C01833=1202.027,168.562,-55.131,-177.976,6.217,148.523
C01834=1202.022,168.811,-55.153,-177.973,6.219,148.522
C01835=1202.018,169.060,-55.175,-177.970,6.220,148.522
C01836=1202.013,169.309,-55.197,-177.968,6.222,148.522
C01837=1202.008,169.559,-55.219,-177.965,6.224,148.521
C01838=1202.003,169.807,-55.241,-177.963,6.225,148.521
C01839=1201.999,170.056,-55.263,-177.960,6.227,148.521
C01840=1201.994,170.305,-55.286,-177.957,6.228,148.520
C01841=1201.990,170.554,-55.308,-177.954,6.230,148.520
C01842=1201.985,170.803,-55.329,-177.952,6.232,148.519
C01843=1201.980,171.052,-55.351,-177.950,6.233,148.519
C01844=1201.975,171.301,-55.374,-177.947,6.235,148.518
C01845=1201.971,171.550,-55.396,-177.944,6.236,148.518
C01846=1201.967,171.799,-55.419,-177.942,6.238,148.518
C01847=1201.962,172.048,-55.440,-177.939,6.240,148.517
C01848=1201.957,172.297,-55.464,-177.936,6.242,148.517
C01849=1201.952,172.546,-55.485,-177.934,6.242,148.516
C01850=1201.948,172.795,-55.507,-177.931,6.244,148.516
C01851=1201.942,173.044,-55.530,-177.928,6.246,148.516
C01852=1201.938,173.293,-55.552,-177.926,6.248,148.515
C01853=1201.934,173.542,-55.574,-177.923,6.250,148.515
C01854=1201.928,173.791,-55.597,-177.920,6.251,148.515
C01855=1201.924,174.040,-55.619,-177.918,6.252,148.514
C01856=1201.920,174.288,-55.641,-177.916,6.254,148.514
C01857=1201.915,174.538,-55.664,-177.913,6.256,148.513
C01858=1201.911,174.787,-55.687,-177.910,6.258,148.513
C01859=1201.906,175.035,-55.708,-177.907,6.259,148.513
C01860=1201.901,175.284,-55.732,-177.904,6.261,148.512
C01861=1201.897,175.534,-55.754,-177.902,6.262,148.512
C01862=1201.891,175.783,-55.776,-177.900,6.264,148.511
C01863=1201.887,176.031,-55.799,-177.897,6.266,148.511
C01864=1201.882,176.280,-55.820,-177.894,6.268,148.511
C01865=1201.878,176.529,-55.844,-177.892,6.269,148.510
C01866=1201.873,176.778,-55.866,-177.889,6.271,148.510
C01867=1201.868,177.027,-55.889,-177.886,6.273,148.510
C01868=1201.864,177.276,-55.911,-177.884,6.274,148.509
C01869=1201.860,177.525,-55.934,-177.882,6.276,148.509
C01870=1201.854,177.774,-55.956,-177.879,6.278,148.509
C01871=1201.850,178.022,-55.979,-177.876,6.279,148.508
C01872=1201.845,178.272,-56.001,-177.873,6.281,148.508
C01873=1201.841,178.520,-56.024,-177.870,6.283,148.507
C01874=1201.836,178.770,-56.046,-177.868,6.284,148.507
C01875=1201.832,179.018,-56.069,-177.866,6.285,148.506
C01876=1201.827,179.268,-56.092,-177.863,6.287,148.506
C01877=1201.822,179.516,-56.114,-177.860,6.289,148.506
C01878=1201.818,179.765,-56.137,-177.858,6.291,148.505
C01879=1201.813,180.014,-56.159,-177.855,6.293,148.505
C01880=1201.808,180.263,-56.182,-177.852,6.294,148.505
C01881=1201.804,180.512,-56.205,-177.850,6.296,148.504
C01882=1201.799,180.761,-56.228,-177.847,6.298,148.504
C01883=1201.795,181.010,-56.251,-177.844,6.300,148.504
C01884=1201.789,181.259,-56.273,-177.842,6.301,148.503
C01885=1201.785,181.508,-56.296,-177.840,6.303,148.503
C01886=1201.781,181.757,-56.319,-177.837,6.304,148.503
C01887=1201.776,182.006,-56.342,-177.834,6.306,148.502
C01888=1201.771,182.254,-56.364,-177.832,6.308,148.502
C01889=1201.766,182.503,-56.387,-177.829,6.310,148.501
C01890=1201.763,182.752,-56.410,-177.826,6.312,148.501
C01891=1201.758,183.002,-56.433,-177.824,6.313,148.501
C01892=1201.752,183.250,-56.456,-177.821,6.315,148.500
C01893=1201.748,183.499,-56.479,-177.818,6.316,148.500
C01894=1201.743,183.748,-56.501,-177.816,6.318,148.499
C01895=1201.739,183.997,-56.524,-177.813,6.320,148.499
C01896=1201.735,184.246,-56.547,-177.810,6.321,148.499
C01897=1201.729,184.494,-56.570,-177.808,6.323,148.498
C01898=1201.725,184.764,-56.595,-177.805,6.325,148.498
C01899=1201.719,185.034,-56.620,-177.802,6.327,148.498
C01900=1201.715,185.303,-56.644,-177.799,6.329,148.497
C01901=1201.709,185.573,-56.669,-177.797,6.331,148.497
C01902=1201.705,185.822,-56.693,-177.794,6.333,148.497
C01903=1201.701,186.071,-56.715,-177.791,6.335,148.496
C01904=1201.696,186.320,-56.739,-177.789,6.336,148.496
C01905=1201.691,186.569,-56.762,-177.787,6.338,148.496
C01906=1201.686,186.817,-56.785,-177.784,6.339,148.495
C01907=1201.682,187.066,-56.807,-177.781,6.341,148.495
C01908=1201.677,187.315,-56.831,-177.778,6.343,148.494
C01909=1201.672,187.564,-56.854,-177.775,6.345,148.494
C01910=1201.668,187.813,-56.877,-177.773,6.346,148.494
C01911=1201.664,188.062,-56.900,-177.770,6.348,148.493
C01912=1201.659,188.311,-56.923,-177.767,6.350,148.493
C01913=1201.654,188.560,-56.946,-177.765,6.352,148.493
C01914=1201.649,188.809,-56.970,-177.762,6.354,148.492
C01915=1201.645,189.057,-56.993,-177.760,6.356,148.492
C01916=1201.640,189.306,-57.016,-177.757,6.358,148.492
C01917=1201.636,189.555,-57.039,-177.755,6.359,148.491
C01918=1201.631,189.804,-57.063,-177.752,6.361,148.491
C01919=1201.626,190.053,-57.086,-177.750,6.362,148.491
C01920=1201.622,190.302,-57.109,-177.747,6.364,148.490
C01921=1201.618,190.551,-57.132,-177.745,6.366,148.490
C01922=1201.612,190.800,-57.155,-177.742,6.368,148.490
C01923=1201.608,191.049,-57.178,-177.739,6.369,148.489
C01924=1201.603,191.298,-57.202,-177.737,6.371,148.489
C01925=1201.599,191.546,-57.226,-177.734,6.373,148.488
C01926=1201.595,191.795,-57.249,-177.731,6.375,148.488
C01927=1201.590,192.044,-57.272,-177.729,6.377,148.488
C01928=1201.585,192.293,-57.295,-177.726,6.378,148.487
C01929=1201.581,192.542,-57.319,-177.723,6.380,148.487
C01930=1201.576,192.791,-57.342,-177.721,6.382,148.487
C01931=1201.571,193.040,-57.365,-177.718,6.384,148.486
C01932=1201.567,193.288,-57.389,-177.715,6.386,148.486
C01933=1201.562,193.537,-57.413,-177.713,6.388,148.486
C01934=1201.557,193.786,-57.436,-177.710,6.389,148.485
C01935=1201.553,194.035,-57.459,-177.707,6.391,148.485
C01936=1201.549,194.284,-57.482,-177.705,6.393,148.485
C01937=1201.544,194.533,-57.506,-177.702,6.395,148.484
C01938=1201.540,194.782,-57.530,-177.699,6.397,148.484
C01939=1201.535,195.031,-57.553,-177.697,6.398,148.484
C01940=1201.530,195.280,-57.576,-177.694,6.400,148.483
C01941=1201.526,195.528,-57.601,-177.691,6.402,148.483
C01942=1201.521,195.777,-57.624,-177.689,6.404,148.483
C01943=1201.516,196.026,-57.647,-177.686,6.406,148.482
C01944=1201.512,196.275,-57.671,-177.683,6.408,148.482
C01945=1201.507,196.524,-57.695,-177.681,6.409,148.482
C01946=1201.503,196.773,-57.718,-177.679,6.411,148.481
C01947=1201.498,197.021,-57.742,-177.676,6.413,148.481
C01948=1201.493,197.270,-57.765,-177.673,6.415,148.481
C01949=1201.489,197.519,-57.789,-177.671,6.417,148.480
C01950=1201.484,197.768,-57.813,-177.668,6.419,148.480
C01951=1201.480,198.017,-57.836,-177.665,6.421,148.480
C01952=1201.475,198.266,-57.860,-177.663,6.422,148.479
C01953=1201.471,198.514,-57.884,-177.660,6.424,148.479
C01954=1201.466,198.763,-57.907,-177.657,6.426,148.479
C01955=1201.461,199.011,-57.931,-177.655,6.428,148.478
C01956=1201.456,199.261,-57.955,-177.652,6.430,148.478
C01957=1201.452,199.509,-57.979,-177.649,6.431,148.478
C01958=1201.447,199.758,-58.003,-177.647,6.433,148.477
C01959=1201.443,200.007,-58.027,-177.644,6.435,148.477
C01960=1201.438,200.256,-58.050,-177.641,6.437,148.477
C01961=1201.433,200.505,-58.073,-177.639,6.439,148.476
C01962=1201.429,200.754,-58.098,-177.637,6.441,148.476
C01963=1201.425,201.002,-58.122,-177.634,6.443,148.476
C01964=1201.420,201.251,-58.145,-177.631,6.445,148.475
C01965=1201.415,201.500,-58.170,-177.629,6.446,148.475
C01966=1201.410,201.749,-58.193,-177.626,6.448,148.475
C01967=1201.406,201.997,-58.217,-177.623,6.450,148.474
C01968=1201.401,202.246,-58.241,-177.621,6.452,148.474
C01969=1201.397,202.495,-58.265,-177.618,6.454,148.474
C01970=1201.392,202.744,-58.288,-177.615,6.455,148.473
C01971=1201.388,202.993,-58.313,-177.613,6.458,148.473
C01972=1201.383,203.242,-58.337,-177.611,6.459,148.473
C01973=1201.379,203.491,-58.361,-177.608,6.461,148.473
C01974=1201.374,203.739,-58.385,-177.605,6.463,148.472
C01975=1201.370,203.988,-58.409,-177.603,6.465,148.472
C01976=1201.364,204.237,-58.433,-177.600,6.467,148.472
C01977=1201.360,204.485,-58.457,-177.597,6.469,148.471
C01978=1201.356,204.734,-58.481,-177.595,6.470,148.471
C01979=1201.352,204.983,-58.505,-177.592,6.472,148.471
C01980=1201.346,205.232,-58.529,-177.589,6.474,148.470
C01981=1201.342,205.481,-58.553,-177.587,6.476,148.470
C01982=1201.338,205.729,-58.577,-177.585,6.478,148.470
C01983=1201.334,205.979,-58.601,-177.582,6.480,148.469
C01984=1201.328,206.228,-58.626,-177.579,6.482,148.469
C01985=1201.324,206.476,-58.650,-177.576,6.484,148.469
C01986=1201.320,206.724,-58.674,-177.573,6.486,148.468
C01987=1201.314,206.974,-58.698,-177.571,6.488,148.468
C01988=1201.310,207.223,-58.722,-177.568,6.490,148.468
C01989=1201.306,207.471,-58.746,-177.566,6.492,148.468
C01990=1201.301,207.720,-58.771,-177.563,6.494,148.467
C01991=1201.296,207.968,-58.795,-177.561,6.496,148.467
C01992=1201.292,208.217,-58.818,-177.558,6.497,148.467
C01993=1201.287,208.467,-58.844,-177.555,6.499,148.466
C01994=1201.283,208.715,-58.868,-177.553,6.501,148.466
C01995=1201.278,208.964,-58.892,-177.550,6.503,148.466
C01996=1201.273,209.212,-58.916,-177.548,6.505,148.465
C01997=1201.269,209.461,-58.941,-177.545,6.507,148.465
C01998=1201.264,209.710,-58.965,-177.543,6.509,148.465
C01999=1201.260,209.959,-58.990,-177.539,6.511,148.464
C02000=1201.256,210.207,-59.014,-177.537,6.513,148.464
C02001=1201.251,210.456,-59.039,-177.534,6.515,148.464
C02002=1201.246,210.727,-59.065,-177.531,6.517,148.463
C02003=1201.241,210.997,-59.091,-177.529,6.519,148.463
C02004=1201.236,211.267,-59.117,-177.526,6.521,148.463
C02005=1201.231,211.538,-59.145,-177.523,6.523,148.462
C02006=1201.226,211.787,-59.169,-177.520,6.525,148.462
C02007=1201.222,212.035,-59.193,-177.518,6.527,148.462
C02008=1201.218,212.284,-59.218,-177.516,6.529,148.462
C02009=1201.213,212.533,-59.242,-177.512,6.532,148.461
C02010=1201.209,212.781,-59.266,-177.510,6.533,148.461
C02011=1201.204,213.031,-59.291,-177.507,6.535,148.461
C02012=1201.200,213.279,-59.316,-177.504,6.537,148.460
C02013=1201.195,213.528,-59.340,-177.502,6.539,148.460
C02014=1201.190,213.776,-59.364,-177.500,6.541,148.460
C02015=1201.186,214.026,-59.389,-177.497,6.543,148.460
C02016=1201.181,214.275,-59.414,-177.494,6.545,148.459
C02017=1201.177,214.524,-59.438,-177.492,6.546,148.459
C02018=1201.172,214.772,-59.464,-177.489,6.549,148.459
C02019=1201.167,215.020,-59.488,-177.486,6.551,148.459
C02020=1201.163,215.270,-59.513,-177.484,6.553,148.458
C02021=1201.159,215.518,-59.537,-177.481,6.555,148.458
C02022=1201.153,215.767,-59.562,-177.478,6.557,148.457
C02023=1201.150,216.016,-59.586,-177.476,6.559,148.457
C02024=1201.145,216.264,-59.612,-177.473,6.561,148.457
C02025=1201.140,216.513,-59.637,-177.471,6.563,148.457
C02026=1201.136,216.762,-59.661,-177.468,6.564,148.456
C02027=1201.131,217.011,-59.685,-177.465,6.567,148.456
C02028=1201.127,217.259,-59.710,-177.462,6.569,148.456
C02029=1201.122,217.508,-59.735,-177.460,6.571,148.456
C02030=1201.118,217.757,-59.760,-177.458,6.573,148.455
C02031=1201.113,218.006,-59.784,-177.455,6.575,148.455
C02032=1201.108,218.254,-59.810,-177.452,6.577,148.455
C02033=1201.104,218.503,-59.835,-177.450,6.578,148.454
C02034=1201.099,218.752,-59.859,-177.447,6.581,148.454
C02035=1201.095,219.000,-59.884,-177.444,6.583,148.454
C02036=1201.090,219.249,-59.909,-177.442,6.585,148.454
C02037=1201.086,219.498,-59.934,-177.439,6.587,148.453
C02038=1201.081,219.746,-59.959,-177.437,6.589,148.453
C02039=1201.076,219.995,-59.984,-177.434,6.591,148.453
C02040=1201.073,220.244,-60.009,-177.432,6.593,148.452
C02041=1201.068,220.492,-60.033,-177.429,6.595,148.452
C02042=1201.063,220.742,-60.058,-177.426,6.597,148.452
C02043=1201.058,220.990,-60.084,-177.424,6.599,148.452
C02044=1201.055,221.239,-60.108,-177.421,6.601,148.451
C02045=1201.050,221.487,-60.134,-177.418,6.603,148.451
C02046=1201.045,221.736,-60.159,-177.416,6.605,148.451
C02047=1201.040,221.985,-60.184,-177.413,6.607,148.451
C02048=1201.037,222.234,-60.209,-177.411,6.609,148.450
C02049=1201.032,222.482,-60.234,-177.408,6.611,148.450
C02050=1201.027,222.731,-60.259,-177.405,6.613,148.450
C02051=1201.022,222.979,-60.284,-177.403,6.615,148.450
C02052=1201.019,223.228,-60.309,-177.400,6.617,148.449
C02053=1201.014,223.476,-60.334,-177.397,6.619,148.449
C02054=1201.009,223.726,-60.359,-177.395,6.621,148.449
C02055=1201.004,223.974,-60.385,-177.392,6.624,148.449
C02056=1201.000,224.223,-60.410,-177.389,6.626,148.448
C02057=1200.995,224.472,-60.435,-177.387,6.628,148.448
C02058=1200.992,224.720,-60.460,-177.384,6.629,148.448
C02059=1200.987,224.969,-60.485,-177.382,6.632,148.447
C02060=1200.982,225.218,-60.511,-177.379,6.633,148.447
C02061=1200.978,225.467,-60.536,-177.376,6.636,148.447
C02062=1200.973,225.715,-60.561,-177.374,6.638,148.447
C02063=1200.969,225.964,-60.587,-177.371,6.640,148.446
C02064=1200.964,226.213,-60.611,-177.369,6.642,148.446
C02065=1200.959,226.461,-60.637,-177.366,6.644,148.446
C02066=1200.954,226.710,-60.663,-177.364,6.646,148.446
C02067=1200.951,226.959,-60.687,-177.361,6.649,148.445
C02068=1200.946,227.207,-60.713,-177.358,6.650,148.445
C02069=1200.942,227.456,-60.738,-177.356,6.653,148.445
C02070=1200.937,227.704,-60.764,-177.353,6.654,148.445
C02071=1200.932,227.953,-60.789,-177.351,6.656,148.444
C02072=1200.928,228.202,-60.814,-177.348,6.658,148.444
C02073=1200.924,228.451,-60.840,-177.345,6.661,148.444
C02074=1200.919,228.699,-60.865,-177.343,6.663,148.443
C02075=1200.914,228.948,-60.891,-177.340,6.665,148.443
C02076=1200.910,229.197,-60.916,-177.338,6.667,148.443
C02077=1200.905,229.445,-60.942,-177.335,6.669,148.443
C02078=1200.901,229.694,-60.967,-177.332,6.671,148.442
C02079=1200.896,229.942,-60.993,-177.330,6.674,148.442
C02080=1200.892,230.191,-61.019,-177.327,6.675,148.442
C02081=1200.888,230.440,-61.044,-177.325,6.677,148.442
C02082=1200.883,230.688,-61.069,-177.322,6.679,148.442
C02083=1200.879,230.937,-61.095,-177.319,6.682,148.441
C02084=1200.874,231.186,-61.120,-177.317,6.684,148.441
C02085=1200.870,231.434,-61.146,-177.314,6.686,148.441
C02086=1200.865,231.683,-61.172,-177.312,6.688,148.441
C02087=1200.861,231.932,-61.197,-177.309,6.690,148.440
C02088=1200.856,232.180,-61.223,-177.306,6.693,148.440
C02089=1200.852,232.429,-61.248,-177.304,6.695,148.440
C02090=1200.847,232.678,-61.275,-177.301,6.696,148.440
C02091=1200.842,232.926,-61.300,-177.299,6.699,148.439
C02092=1200.838,233.175,-61.326,-177.296,6.700,148.439
C02093=1200.834,233.423,-61.352,-177.293,6.703,148.439
C02094=1200.830,233.672,-61.377,-177.291,6.705,148.439
C02095=1200.825,233.920,-61.403,-177.288,6.707,148.438
C02096=1200.821,234.169,-61.429,-177.286,6.709,148.438
C02097=1200.816,234.418,-61.454,-177.284,6.711,148.438
C02098=1200.811,234.666,-61.480,-177.280,6.714,148.438
C02099=1200.807,234.915,-61.506,-177.278,6.716,148.437
C02100=1200.802,235.164,-61.532,-177.276,6.718,148.437
C02101=1200.798,235.413,-61.558,-177.273,6.720,148.437
C02102=1200.793,235.661,-61.583,-177.270,6.722,148.437
C02103=1200.789,235.910,-61.609,-177.268,6.724,148.437
C02104=1200.784,236.159,-61.635,-177.265,6.726,148.436
C02105=1200.780,236.408,-61.661,-177.263,6.728,148.436
C02106=1200.775,236.678,-61.689,-177.260,6.731,148.436
C02107=1200.770,236.950,-61.717,-177.257,6.733,148.436
C02108=1200.766,237.221,-61.746,-177.254,6.736,148.435
C02109=1200.760,237.493,-61.774,-177.251,6.738,148.435
C02110=1200.755,237.742,-61.800,-177.248,6.741,148.435
C02111=1200.751,237.990,-61.826,-177.246,6.742,148.435
C02112=1200.747,238.239,-61.852,-177.244,6.745,148.434
C02113=1200.742,238.488,-61.879,-177.241,6.746,148.434
C02114=1200.738,238.736,-61.904,-177.238,6.749,148.434
C02115=1200.733,238.985,-61.930,-177.236,6.751,148.434
C02116=1200.729,239.233,-61.956,-177.233,6.753,148.433
C02117=1200.724,239.482,-61.983,-177.231,6.755,148.433
C02118=1200.720,239.731,-62.008,-177.228,6.758,148.433
C02119=1200.716,239.978,-62.034,-177.225,6.760,148.433
C02120=1200.711,240.227,-62.061,-177.223,6.762,148.433
C02121=1200.707,240.476,-62.086,-177.220,6.764,148.432
C02122=1200.703,240.724,-62.113,-177.218,6.767,148.432
C02123=1200.698,240.974,-62.139,-177.215,6.769,148.432
C02124=1200.693,241.222,-62.165,-177.212,6.770,148.432
C02125=1200.690,241.471,-62.192,-177.210,6.773,148.432
C02126=1200.684,241.719,-62.217,-177.207,6.775,148.431
C02127=1200.680,241.968,-62.243,-177.205,6.777,148.431
C02128=1200.675,242.216,-62.270,-177.202,6.779,148.431
C02129=1200.671,242.465,-62.296,-177.200,6.781,148.431
C02130=1200.667,242.713,-62.323,-177.197,6.784,148.430
C02131=1200.662,242.962,-62.349,-177.194,6.786,148.430
C02132=1200.658,243.211,-62.375,-177.192,6.788,148.430
C02133=1200.653,243.460,-62.402,-177.189,6.791,148.430
C02134=1200.648,243.708,-62.427,-177.187,6.793,148.430
C02135=1200.644,243.956,-62.454,-177.184,6.795,148.429
C02136=1200.639,244.205,-62.480,-177.182,6.797,148.429
C02137=1200.635,244.453,-62.506,-177.179,6.800,148.429
C02138=1200.631,244.702,-62.533,-177.177,6.802,148.429
C02139=1200.627,244.951,-62.559,-177.174,6.804,148.429
C02140=1200.622,245.199,-62.586,-177.171,6.806,148.428
C02141=1200.618,245.448,-62.612,-177.169,6.809,148.428
C02142=1200.613,245.696,-62.639,-177.166,6.810,148.428
C02143=1200.609,245.945,-62.665,-177.164,6.813,148.428
C02144=1200.604,246.194,-62.692,-177.161,6.815,148.427
C02145=1200.600,246.442,-62.718,-177.158,6.817,148.427
C02146=1200.595,246.691,-62.745,-177.156,6.819,148.427
C02147=1200.591,246.939,-62.771,-177.153,6.822,148.427
C02148=1200.586,247.188,-62.797,-177.150,6.824,148.427
C02149=1200.582,247.436,-62.824,-177.148,6.826,148.427
C02150=1200.578,247.685,-62.851,-177.146,6.828,148.426
C02151=1200.573,247.933,-62.876,-177.143,6.831,148.426
C02152=1200.568,248.181,-62.903,-177.140,6.833,148.426
C02153=1200.564,248.430,-62.930,-177.138,6.835,148.426
C02154=1200.559,248.679,-62.956,-177.135,6.838,148.426
C02155=1200.555,248.927,-62.983,-177.132,6.840,148.425
C02156=1200.551,249.175,-63.010,-177.130,6.842,148.425
C02157=1200.546,249.424,-63.037,-177.127,6.844,148.425
C02158=1200.541,249.673,-63.063,-177.125,6.847,148.425
C02159=1200.537,249.921,-63.090,-177.122,6.848,148.424
C02160=1200.533,250.170,-63.117,-177.120,6.851,148.424
C02161=1200.529,250.419,-63.144,-177.117,6.853,148.424
C02162=1200.525,250.667,-63.171,-177.115,6.855,148.424
C02163=1200.520,250.916,-63.197,-177.112,6.858,148.424
C02164=1200.516,251.164,-63.223,-177.109,6.860,148.424
C02165=1200.511,251.413,-63.250,-177.107,6.862,148.423
C02166=1200.506,251.661,-63.278,-177.104,6.865,148.423
C02167=1200.502,251.910,-63.305,-177.101,6.867,148.423
C02168=1200.498,252.158,-63.331,-177.099,6.869,148.423
C02169=1200.493,252.407,-63.358,-177.097,6.872,148.423
C02170=1200.488,252.656,-63.384,-177.094,6.874,148.423
C02171=1200.484,252.904,-63.411,-177.092,6.876,148.422
C02172=1200.480,253.152,-63.438,-177.089,6.879,148.422
C02173=1200.475,253.401,-63.465,-177.086,6.881,148.422
C02174=1200.470,253.649,-63.492,-177.084,6.883,148.422
C02175=1200.466,253.898,-63.519,-177.081,6.886,148.422
C02176=1200.462,254.147,-63.546,-177.079,6.888,148.421
C02177=1200.458,254.395,-63.573,-177.076,6.890,148.421
C02178=1200.453,254.644,-63.600,-177.073,6.893,148.421
C02179=1200.449,254.892,-63.627,-177.071,6.895,148.421
C02180=1200.445,255.140,-63.654,-177.068,6.897,148.421
C02181=1200.440,255.389,-63.681,-177.066,6.900,148.421
C02182=1200.435,255.637,-63.708,-177.063,6.902,148.420
C02183=1200.431,255.886,-63.735,-177.061,6.904,148.420
C02184=1200.427,256.134,-63.761,-177.058,6.907,148.420
C02185=1200.423,256.383,-63.789,-177.056,6.909,148.420
C02186=1200.418,256.632,-63.816,-177.053,6.912,148.420
C02187=1200.414,256.880,-63.844,-177.050,6.913,148.419
C02188=1200.409,257.128,-63.871,-177.048,6.916,148.419
C02189=1200.404,257.377,-63.898,-177.045,6.918,148.419
C02190=1200.400,257.625,-63.924,-177.043,6.920,148.419
C02191=1200.396,257.874,-63.952,-177.040,6.922,148.419
C02192=1200.392,258.123,-63.979,-177.037,6.925,148.419
C02193=1200.387,258.371,-64.006,-177.035,6.927,148.419
C02194=1200.383,258.619,-64.033,-177.032,6.930,148.418
C02195=1200.378,258.867,-64.061,-177.030,6.932,148.418
C02196=1200.373,259.116,-64.088,-177.027,6.934,148.418
C02197=1200.369,259.365,-64.115,-177.025,6.937,148.418
C02198=1200.365,259.614,-64.142,-177.022,6.939,148.418
C02199=1200.360,259.861,-64.170,-177.019,6.942,148.418
C02200=1200.356,260.110,-64.197,-177.017,6.944,148.417
C02201=1200.352,260.359,-64.224,-177.014,6.946,148.417
C02202=1200.348,260.607,-64.252,-177.012,6.949,148.417
C02203=1200.343,260.855,-64.279,-177.009,6.951,148.417
C02204=1200.339,261.104,-64.306,-177.006,6.954,148.417
C02205=1200.334,261.352,-64.333,-177.004,6.956,148.417
C02206=1200.330,261.601,-64.361,-177.002,6.958,148.416
C02207=1200.326,261.849,-64.388,-176.999,6.961,148.416
C02208=1200.321,262.098,-64.415,-176.996,6.963,148.416
C02209=1200.317,262.346,-64.443,-176.994,6.966,148.416
C02210=1200.312,262.619,-64.473,-176.991,6.968,148.416
C02211=1200.307,262.892,-64.504,-176.988,6.971,148.416
C02212=1200.302,263.164,-64.533,-176.985,6.973,148.415
C02213=1200.297,263.438,-64.563,-176.982,6.976,148.415
C02214=1200.293,263.686,-64.591,-176.980,6.979,148.415
C02215=1200.288,263.934,-64.618,-176.978,6.980,148.415
C02216=1200.284,264.183,-64.646,-176.975,6.983,148.415
C02217=1200.280,264.431,-64.673,-176.972,6.985,148.415
C02218=1200.275,264.679,-64.701,-176.970,6.988,148.415
C02219=1200.271,264.928,-64.729,-176.967,6.990,148.414
C02220=1200.267,265.176,-64.756,-176.965,6.992,148.414
C02221=1200.262,265.425,-64.784,-176.962,6.995,148.414
C02222=1200.257,265.673,-64.812,-176.960,6.997,148.414
C02223=1200.253,265.922,-64.839,-176.957,7.000,148.414
C02224=1200.249,266.170,-64.867,-176.955,7.002,148.414
C02225=1200.244,266.419,-64.894,-176.952,7.005,148.414
C02226=1200.240,266.667,-64.922,-176.949,7.007,148.413
C02227=1200.236,266.915,-64.950,-176.947,7.010,148.413
C02228=1200.231,267.164,-64.978,-176.944,7.012,148.413
C02229=1200.227,267.412,-65.006,-176.942,7.014,148.413
C02230=1200.222,267.661,-65.033,-176.939,7.017,148.413
C02231=1200.219,267.909,-65.061,-176.937,7.019,148.413
C02232=1200.214,268.157,-65.089,-176.934,7.022,148.413
C02233=1200.209,268.406,-65.117,-176.932,7.024,148.412
C02234=1200.205,268.655,-65.145,-176.929,7.027,148.412
C02235=1200.201,268.903,-65.172,-176.926,7.029,148.412
C02236=1200.196,269.151,-65.200,-176.924,7.032,148.412
C02237=1200.192,269.400,-65.228,-176.921,7.034,148.412
C02238=1200.187,269.648,-65.256,-176.919,7.036,148.412
C02239=1200.183,269.896,-65.284,-176.916,7.039,148.412
C02240=1200.179,270.145,-65.311,-176.914,7.041,148.412
C02241=1200.174,270.393,-65.340,-176.911,7.044,148.411
C02242=1200.170,270.642,-65.368,-176.909,7.046,148.411
C02243=1200.166,270.890,-65.396,-176.906,7.049,148.411
C02244=1200.162,271.139,-65.423,-176.903,7.051,148.411
C02245=1200.156,271.387,-65.451,-176.901,7.054,148.411
C02246=1200.152,271.635,-65.479,-176.899,7.056,148.411
C02247=1200.148,271.883,-65.507,-176.895,7.059,148.411
C02248=1200.143,272.132,-65.536,-176.893,7.061,148.410
C02249=1200.139,272.381,-65.563,-176.891,7.064,148.410
C02250=1200.135,272.629,-65.591,-176.888,7.066,148.410
C02251=1200.130,272.878,-65.620,-176.885,7.069,148.410
C02252=1200.126,273.125,-65.647,-176.883,7.071,148.410
C02253=1200.122,273.374,-65.675,-176.880,7.074,148.410
C02254=1200.117,273.622,-65.704,-176.878,7.076,148.410
C02255=1200.113,273.871,-65.732,-176.875,7.079,148.410
C02256=1200.108,274.119,-65.760,-176.873,7.081,148.410
C02257=1200.105,274.367,-65.789,-176.871,7.083,148.409
C02258=1200.100,274.615,-65.816,-176.868,7.086,148.409
C02259=1200.096,274.864,-65.845,-176.865,7.088,148.409
C02260=1200.091,275.112,-65.873,-176.863,7.091,148.409
C02261=1200.087,275.361,-65.902,-176.860,7.093,148.409
C02262=1200.083,275.609,-65.929,-176.857,7.096,148.409
C02263=1200.079,275.857,-65.957,-176.855,7.098,148.409
C02264=1200.074,276.106,-65.986,-176.853,7.101,148.409
C02265=1200.070,276.354,-66.014,-176.850,7.103,148.408
C02266=1200.065,276.602,-66.042,-176.847,7.106,148.408
C02267=1200.061,276.851,-66.070,-176.845,7.108,148.408
C02268=1200.056,277.099,-66.099,-176.842,7.111,148.408
C02269=1200.052,277.348,-66.127,-176.839,7.114,148.408
C02270=1200.047,277.596,-66.155,-176.837,7.116,148.408
C02271=1200.043,277.845,-66.184,-176.834,7.119,148.408
C02272=1200.039,278.093,-66.212,-176.832,7.122,148.408
C02273=1200.035,278.341,-66.241,-176.829,7.124,148.408
C02274=1200.030,278.590,-66.269,-176.827,7.126,148.407
C02275=1200.026,278.837,-66.297,-176.824,7.129,148.407
C02276=1200.022,279.086,-66.326,-176.822,7.132,148.407
C02277=1200.017,279.334,-66.354,-176.819,7.135,148.407
C02278=1200.013,279.583,-66.383,-176.817,7.136,148.407
C02279=1200.009,279.831,-66.412,-176.814,7.139,148.407
C02280=1200.004,280.079,-66.440,-176.812,7.142,148.407
C02281=1200.000,280.328,-66.468,-176.809,7.145,148.407
C02282=1199.995,280.576,-66.496,-176.807,7.147,148.407
C02283=1199.991,280.824,-66.526,-176.804,7.150,148.407
C02284=1199.987,281.073,-66.554,-176.802,7.152,148.407
C02285=1199.982,281.321,-66.582,-176.799,7.155,148.406
C02286=1199.978,281.569,-66.612,-176.797,7.157,148.406
C02287=1199.974,281.818,-66.640,-176.794,7.160,148.406
C02288=1199.969,282.066,-66.668,-176.791,7.163,148.406
C02289=1199.965,282.314,-66.698,-176.789,7.165,148.406
C02290=1199.961,282.562,-66.725,-176.786,7.168,148.406
C02291=1199.956,282.811,-66.754,-176.784,7.170,148.406
C02292=1199.952,283.059,-66.784,-176.781,7.173,148.406
C02293=1199.948,283.307,-66.811,-176.779,7.175,148.406
C02294=1199.943,283.556,-66.840,-176.776,7.178,148.406
C02295=1199.939,283.804,-66.870,-176.774,7.180,148.406
C02296=1199.935,284.052,-66.897,-176.771,7.183,148.405
C02297=1199.931,284.301,-66.927,-176.769,7.185,148.405
C02298=1199.926,284.549,-66.956,-176.766,7.188,148.405
C02299=1199.921,284.797,-66.985,-176.763,7.191,148.405
C02300=1199.918,285.046,-67.013,-176.761,7.193,148.405
C02301=1199.913,285.294,-67.042,-176.758,7.196,148.405
C02302=1199.909,285.543,-67.071,-176.756,7.198,148.405
C02303=1199.904,285.790,-67.100,-176.753,7.201,148.405
C02304=1199.900,286.039,-67.128,-176.751,7.204,148.405
C02305=1199.896,286.287,-67.158,-176.748,7.206,148.405
C02306=1199.891,286.535,-67.186,-176.745,7.209,148.405
C02307=1199.887,286.784,-67.215,-176.743,7.211,148.405
C02308=1199.882,287.032,-67.244,-176.741,7.214,148.405
C02309=1199.879,287.280,-67.273,-176.738,7.217,148.404
C02310=1199.874,287.529,-67.301,-176.736,7.220,148.404
C02311=1199.870,287.777,-67.331,-176.734,7.222,148.404
C02312=1199.866,288.025,-67.360,-176.730,7.225,148.404
C02313=1199.861,288.274,-67.389,-176.728,7.228,148.404
C02314=1199.857,288.548,-67.421,-176.726,7.230,148.404
C02315=1199.852,288.822,-67.453,-176.723,7.233,148.404
C02316=1199.846,289.097,-67.485,-176.720,7.236,148.404
C02317=1199.842,289.371,-67.518,-176.717,7.238,148.404
C02318=1199.837,289.619,-67.546,-176.714,7.241,148.404
C02319=1199.833,289.868,-67.576,-176.712,7.244,148.404
C02320=1199.829,290.116,-67.605,-176.710,7.247,148.404
C02321=1199.825,290.364,-67.634,-176.707,7.250,148.404
C02322=1199.820,290.612,-67.663,-176.705,7.252,148.404
C02323=1199.816,290.860,-67.692,-176.702,7.255,148.403
C02324=1199.812,291.109,-67.721,-176.700,7.257,148.403
C02325=1199.808,291.357,-67.751,-176.697,7.260,148.403
C02326=1199.803,291.606,-67.780,-176.694,7.263,148.403
C02327=1199.799,291.854,-67.809,-176.692,7.265,148.403
C02328=1199.794,292.102,-67.838,-176.689,7.268,148.403
C02329=1199.790,292.350,-67.868,-176.687,7.270,148.403
C02330=1199.786,292.598,-67.897,-176.684,7.273,148.403
C02331=1199.782,292.846,-67.927,-176.682,7.276,148.403
C02332=1199.778,293.095,-67.956,-176.679,7.278,148.403
C02333=1199.773,293.344,-67.985,-176.677,7.281,148.403
C02334=1199.768,293.591,-68.014,-176.674,7.284,148.403
C02335=1199.764,293.839,-68.043,-176.672,7.287,148.403
C02336=1199.760,294.088,-68.073,-176.669,7.290,148.403
C02337=1199.756,294.336,-68.102,-176.667,7.292,148.403
C02338=1199.752,294.584,-68.132,-176.664,7.295,148.403
C02339=1199.747,294.832,-68.161,-176.662,7.298,148.403
C02340=1199.743,295.081,-68.191,-176.660,7.300,148.403
C02341=1199.739,295.329,-68.220,-176.657,7.303,148.403
C02342=1199.735,295.577,-68.249,-176.654,7.305,148.402
C02343=1199.731,295.826,-68.279,-176.652,7.308,148.402
C02344=1199.726,296.073,-68.308,-176.649,7.311,148.402
C02345=1199.721,296.322,-68.338,-176.647,7.313,148.402
C02346=1199.717,296.570,-68.368,-176.644,7.316,148.402
C02347=1199.713,296.818,-68.397,-176.641,7.319,148.402
C02348=1199.708,297.066,-68.426,-176.639,7.321,148.402
C02349=1199.704,297.315,-68.456,-176.637,7.324,148.402
C02350=1199.700,297.563,-68.485,-176.634,7.327,148.402
C02351=1199.696,297.811,-68.515,-176.632,7.330,148.402
C02352=1199.692,298.059,-68.545,-176.629,7.333,148.402
C02353=1199.687,298.308,-68.575,-176.627,7.335,148.402
C02354=1199.683,298.556,-68.604,-176.624,7.338,148.402
C02355=1199.679,298.804,-68.634,-176.621,7.341,148.402
C02356=1199.675,299.052,-68.663,-176.619,7.343,148.402
C02357=1199.670,299.301,-68.693,-176.617,7.346,148.402
C02358=1199.666,299.549,-68.724,-176.614,7.348,148.402
C02359=1199.662,299.797,-68.753,-176.612,7.351,148.402
C02360=1199.657,300.045,-68.782,-176.609,7.354,148.402
C02361=1199.653,300.293,-68.812,-176.607,7.356,148.402
C02362=1199.649,300.541,-68.842,-176.604,7.359,148.402
C02363=1199.644,300.790,-68.872,-176.602,7.362,148.402
C02364=1199.640,301.038,-68.902,-176.600,7.365,148.402
C02365=1199.636,301.286,-68.931,-176.597,7.368,148.402
C02366=1199.631,301.534,-68.962,-176.594,7.371,148.402
C02367=1199.627,301.782,-68.991,-176.592,7.373,148.402
C02368=1199.623,302.031,-69.021,-176.590,7.376,148.402
C02369=1199.619,302.278,-69.051,-176.587,7.379,148.402
C02370=1199.614,302.527,-69.081,-176.585,7.381,148.402
C02371=1199.610,302.775,-69.110,-176.582,7.384,148.402
C02372=1199.606,303.023,-69.141,-176.579,7.387,148.401
C02373=1199.601,303.271,-69.171,-176.577,7.390,148.401
C02374=1199.597,303.519,-69.201,-176.575,7.393,148.401
C02375=1199.593,303.767,-69.230,-176.572,7.396,148.401
C02376=1199.588,304.016,-69.260,-176.570,7.398,148.401
C02377=1199.584,304.263,-69.290,-176.567,7.401,148.401
C02378=1199.580,304.512,-69.320,-176.564,7.404,148.401
C02379=1199.576,304.760,-69.351,-176.562,7.406,148.401
C02380=1199.571,305.008,-69.380,-176.560,7.409,148.401
C02381=1199.567,305.256,-69.411,-176.558,7.412,148.401
C02382=1199.563,305.505,-69.441,-176.555,7.415,148.401
C02383=1199.559,305.753,-69.471,-176.553,7.418,148.401
C02384=1199.554,306.001,-69.501,-176.550,7.420,148.401
C02385=1199.551,306.249,-69.531,-176.548,7.423,148.401
C02386=1199.546,306.497,-69.561,-176.545,7.426,148.401
C02387=1199.542,306.745,-69.591,-176.543,7.428,148.401
C02388=1199.537,306.994,-69.621,-176.540,7.431,148.401
C02389=1199.533,307.241,-69.652,-176.538,7.434,148.401
C02390=1199.528,307.489,-69.682,-176.535,7.437,148.401
C02391=1199.525,307.738,-69.712,-176.533,7.440,148.401
C02392=1199.520,307.986,-69.743,-176.530,7.443,148.401
C02393=1199.516,308.234,-69.772,-176.528,7.446,148.401
C02394=1199.511,308.482,-69.803,-176.526,7.448,148.401
C02395=1199.508,308.730,-69.833,-176.523,7.451,148.401
C02396=1199.503,308.979,-69.863,-176.521,7.454,148.401
C02397=1199.499,309.226,-69.893,-176.519,7.456,148.401
C02398=1199.495,309.475,-69.925,-176.516,7.459,148.401
C02399=1199.491,309.723,-69.954,-176.513,7.462,148.401
C02400=1199.486,309.971,-69.985,-176.511,7.465,148.401
C02401=1199.482,310.219,-70.015,-176.508,7.468,148.401
C02402=1199.477,310.467,-70.046,-176.506,7.471,148.402
C02403=1199.474,310.716,-70.076,-176.504,7.473,148.401
C02404=1199.469,310.964,-70.106,-176.501,7.476,148.401
C02405=1199.465,311.212,-70.137,-176.499,7.479,148.401
C02406=1199.461,311.459,-70.167,-176.496,7.481,148.401
C02407=1199.456,311.707,-70.198,-176.494,7.485,148.402
C02408=1199.453,311.956,-70.228,-176.492,7.488,148.402
C02409=1199.448,312.204,-70.259,-176.489,7.490,148.402
C02410=1199.443,312.452,-70.289,-176.487,7.493,148.402
C02411=1199.439,312.700,-70.320,-176.484,7.496,148.401
C02412=1199.435,312.948,-70.350,-176.482,7.499,148.402
C02413=1199.431,313.196,-70.381,-176.480,7.502,148.402
C02414=1199.427,313.444,-70.412,-176.477,7.505,148.402
C02415=1199.422,313.692,-70.442,-176.474,7.508,148.402
C02416=1199.417,313.940,-70.472,-176.473,7.510,148.402
C02417=1199.414,314.189,-70.503,-176.470,7.513,148.402
C02418=1199.409,314.465,-70.537,-176.467,7.516,148.402
C02419=1199.405,314.740,-70.572,-176.464,7.519,148.402
C02420=1199.400,315.018,-70.605,-176.462,7.522,148.402
C02421=1199.395,315.293,-70.640,-176.459,7.526,148.402
C02422=1199.391,315.541,-70.670,-176.457,7.529,148.402
C02423=1199.387,315.790,-70.702,-176.454,7.532,148.402
C02424=1199.382,316.038,-70.732,-176.452,7.535,148.402
C02425=1199.378,316.286,-70.763,-176.450,7.537,148.402
C02426=1199.374,316.534,-70.794,-176.447,7.540,148.402
C02427=1199.370,316.782,-70.824,-176.444,7.543,148.402
C02428=1199.365,317.030,-70.855,-176.442,7.545,148.402
C02429=1199.362,317.278,-70.886,-176.440,7.549,148.402
C02430=1199.357,317.526,-70.917,-176.437,7.552,148.402
C02431=1199.352,317.774,-70.947,-176.435,7.555,148.402
C02432=1199.349,318.022,-70.979,-176.433,7.557,148.402
C02433=1199.344,318.270,-71.010,-176.430,7.560,148.402
C02434=1199.340,318.518,-71.040,-176.428,7.563,148.402
C02435=1199.336,318.767,-71.071,-176.426,7.566,148.403
C02436=1199.332,319.015,-71.102,-176.423,7.569,148.403
C02437=1199.327,319.263,-71.133,-176.421,7.572,148.403
C02438=1199.323,319.511,-71.165,-176.418,7.575,148.403
C02439=1199.319,319.758,-71.195,-176.416,7.577,148.403
C02440=1199.315,320.006,-71.225,-176.414,7.580,148.403
C02441=1199.311,320.255,-71.257,-176.411,7.584,148.403
C02442=1199.307,320.502,-71.288,-176.409,7.586,148.403
C02443=1199.303,320.751,-71.319,-176.407,7.589,148.403
C02444=1199.298,320.999,-71.350,-176.404,7.592,148.403
C02445=1199.293,321.247,-71.381,-176.402,7.595,148.403
C02446=1199.290,321.495,-71.413,-176.399,7.597,148.403
C02447=1199.285,321.743,-71.443,-176.397,7.601,148.403
C02448=1199.281,321.992,-71.474,-176.395,7.604,148.403
C02449=1199.277,322.239,-71.505,-176.393,7.606,148.403
C02450=1199.273,322.486,-71.536,-176.390,7.609,148.403
C02451=1199.269,322.735,-71.567,-176.387,7.612,148.403
C02452=1199.264,322.982,-71.599,-176.385,7.616,148.404
C02453=1199.260,323.231,-71.630,-176.383,7.618,148.404
C02454=1199.256,323.478,-71.661,-176.381,7.621,148.404
C02455=1199.252,323.727,-71.692,-176.378,7.624,148.404
C02456=1199.248,323.975,-71.723,-176.376,7.626,148.404
C02457=1199.244,324.223,-71.755,-176.374,7.630,148.404
C02458=1199.239,324.471,-71.786,-176.371,7.633,148.404
C02459=1199.235,324.719,-71.818,-176.369,7.636,148.404
C02460=1199.231,324.967,-71.848,-176.367,7.638,148.404
C02461=1199.227,325.215,-71.880,-176.365,7.642,148.404
C02462=1199.223,325.463,-71.911,-176.362,7.645,148.404
C02463=1199.219,325.711,-71.943,-176.360,7.647,148.404
C02464=1199.214,325.959,-71.974,-176.358,7.650,148.404
C02465=1199.211,326.207,-72.006,-176.355,7.654,148.405
C02466=1199.206,326.455,-72.036,-176.353,7.657,148.405
C02467=1199.201,326.703,-72.069,-176.351,7.659,148.405
C02468=1199.197,326.951,-72.100,-176.348,7.662,148.405
C02469=1199.193,327.199,-72.131,-176.346,7.665,148.405
C02470=1199.189,327.447,-72.163,-176.343,7.668,148.405
C02471=1199.185,327.695,-72.194,-176.342,7.671,148.405
C02472=1199.181,327.943,-72.225,-176.339,7.674,148.405
C02473=1199.177,328.191,-72.257,-176.337,7.677,148.405
C02474=1199.172,328.439,-72.288,-176.335,7.679,148.405
C02475=1199.169,328.687,-72.320,-176.332,7.683,148.406
C02476=1199.163,328.934,-72.352,-176.330,7.686,148.406
C02477=1199.159,329.183,-72.383,-176.327,7.689,148.406
C02478=1199.155,329.430,-72.415,-176.325,7.691,148.406
C02479=1199.151,329.678,-72.446,-176.323,7.695,148.406
C02480=1199.147,329.926,-72.477,-176.320,7.698,148.406
C02481=1199.143,330.174,-72.509,-176.318,7.701,148.406
C02482=1199.139,330.423,-72.541,-176.316,7.703,148.406
C02483=1199.134,330.670,-72.573,-176.314,7.707,148.406
C02484=1199.130,330.919,-72.604,-176.312,7.710,148.407
C02485=1199.126,331.166,-72.636,-176.310,7.712,148.407
C02486=1199.122,331.415,-72.668,-176.307,7.715,148.407
C02487=1199.118,331.663,-72.700,-176.305,7.719,148.407
C02488=1199.114,331.910,-72.731,-176.302,7.722,148.407
C02489=1199.110,332.159,-72.762,-176.301,7.724,148.407
C02490=1199.105,332.406,-72.795,-176.298,7.727,148.407
C02491=1199.101,332.654,-72.826,-176.296,7.731,148.407
C02492=1199.097,332.902,-72.858,-176.294,7.734,148.408
C02493=1199.093,333.150,-72.890,-176.291,7.736,148.408
C02494=1199.088,333.398,-72.922,-176.289,7.740,148.408
C02495=1199.084,333.645,-72.954,-176.287,7.743,148.408
C02496=1199.080,333.893,-72.985,-176.285,7.745,148.408
C02497=1199.076,334.142,-73.017,-176.283,7.748,148.408
C02498=1199.071,334.390,-73.049,-176.280,7.751,148.408
C02499=1199.068,334.638,-73.081,-176.278,7.755,148.408
C02500=1199.063,334.886,-73.113,-176.276,7.757,148.409
C02501=1199.059,335.133,-73.144,-176.273,7.760,148.409
C02502=1199.055,335.381,-73.176,-176.271,7.764,148.409
C02503=1199.051,335.630,-73.209,-176.269,7.767,148.409
C02504=1199.046,335.877,-73.240,-176.267,7.769,148.409
C02505=1199.043,336.125,-73.272,-176.265,7.773,148.409
C02506=1199.038,336.373,-73.304,-176.262,7.776,148.409
C02507=1199.034,336.621,-73.336,-176.261,7.778,148.410
C02508=1199.030,336.869,-73.369,-176.258,7.781,148.410
C02509=1199.026,337.117,-73.401,-176.256,7.785,148.410
C02510=1199.022,337.365,-73.433,-176.253,7.788,148.410
C02511=1199.017,337.612,-73.465,-176.252,7.791,148.410
C02512=1199.014,337.860,-73.497,-176.249,7.794,148.410
C02513=1199.009,338.109,-73.529,-176.247,7.797,148.410
C02514=1199.005,338.356,-73.561,-176.245,7.800,148.411
C02515=1199.000,338.604,-73.593,-176.243,7.803,148.411
C02516=1198.997,338.852,-73.626,-176.241,7.806,148.411
C02517=1198.993,339.100,-73.658,-176.238,7.809,148.411
C02518=1198.988,339.347,-73.690,-176.236,7.812,148.411
C02519=1198.985,339.595,-73.721,-176.234,7.815,148.411
C02520=1198.980,339.844,-73.754,-176.232,7.818,148.412
C02521=1198.977,340.091,-73.786,-176.230,7.822,148.412
C02522=1198.971,340.370,-73.822,-176.227,7.825,148.412
C02523=1198.967,340.648,-73.858,-176.225,7.828,148.412
C02524=1198.962,340.927,-73.895,-176.223,7.831,148.412
C02525=1198.957,341.205,-73.931,-176.220,7.835,148.413
C02526=1198.953,341.453,-73.964,-176.218,7.838,148.413
C02527=1198.949,341.701,-73.996,-176.216,7.841,148.413
C02528=1198.945,341.949,-74.029,-176.214,7.845,148.413
C02529=1198.941,342.196,-74.060,-176.212,7.847,148.413
C02530=1198.936,342.444,-74.093,-176.209,7.850,148.413
C02531=1198.932,342.692,-74.126,-176.207,7.854,148.414
C02532=1198.929,342.940,-74.158,-176.205,7.857,148.414
C02533=1198.924,343.189,-74.190,-176.203,7.859,148.414
C02534=1198.920,343.435,-74.222,-176.201,7.863,148.414
C02535=1198.916,343.684,-74.255,-176.199,7.866,148.414
C02536=1198.911,343.932,-74.287,-176.197,7.869,148.415
C02537=1198.908,344.179,-74.320,-176.195,7.872,148.415
C02538=1198.903,344.428,-74.352,-176.193,7.875,148.415
C02539=1198.899,344.675,-74.385,-176.190,7.879,148.415
C02540=1198.895,344.923,-74.417,-176.189,7.881,148.415
C02541=1198.891,345.171,-74.450,-176.187,7.884,148.416
C02542=1198.886,345.419,-74.482,-176.184,7.888,148.416
C02543=1198.883,345.666,-74.515,-176.183,7.890,148.416
C02544=1198.878,345.915,-74.547,-176.180,7.894,148.416
C02545=1198.874,346.162,-74.581,-176.178,7.897,148.416
C02546=1198.870,346.410,-74.612,-176.176,7.900,148.417
C02547=1198.866,346.658,-74.645,-176.174,7.903,148.417
C02548=1198.861,346.906,-74.678,-176.172,7.906,148.417
C02549=1198.857,347.154,-74.711,-176.170,7.909,148.417
C02550=1198.854,347.402,-74.743,-176.168,7.913,148.418
C02551=1198.849,347.649,-74.776,-176.166,7.915,148.418
C02552=1198.845,347.897,-74.809,-176.164,7.919,148.418
C02553=1198.841,348.145,-74.841,-176.161,7.922,148.418
C02554=1198.837,348.393,-74.874,-176.160,7.924,148.418
C02555=1198.833,348.640,-74.907,-176.158,7.928,148.419
C02556=1198.828,348.888,-74.939,-176.155,7.931,148.419
C02557=1198.824,349.136,-74.972,-176.153,7.934,148.419
C02558=1198.821,349.383,-75.005,-176.151,7.937,148.419
C02559=1198.816,349.632,-75.037,-176.150,7.941,148.420
C02560=1198.812,349.879,-75.070,-176.147,7.944,148.420
C02561=1198.808,350.127,-75.104,-176.146,7.946,148.420
C02562=1198.804,350.376,-75.136,-176.144,7.950,148.420
C02563=1198.800,350.623,-75.169,-176.141,7.953,148.420
C02564=1198.796,350.871,-75.202,-176.139,7.956,148.421
C02565=1198.792,351.118,-75.235,-176.137,7.959,148.421
C02566=1198.787,351.367,-75.267,-176.136,7.963,148.421
C02567=1198.783,351.614,-75.301,-176.133,7.966,148.422
C02568=1198.779,351.862,-75.334,-176.132,7.968,148.422
C02569=1198.775,352.110,-75.367,-176.129,7.972,148.422
C02570=1198.772,352.357,-75.399,-176.127,7.975,148.422
C02571=1198.767,352.606,-75.432,-176.126,7.978,148.423
C02572=1198.763,352.853,-75.465,-176.124,7.981,148.423
C02573=1198.759,353.101,-75.498,-176.122,7.985,148.423
C02574=1198.755,353.349,-75.531,-176.119,7.988,148.423
C02575=1198.751,353.597,-75.564,-176.118,7.991,148.424
C02576=1198.747,353.844,-75.598,-176.116,7.994,148.424
C02577=1198.742,354.092,-75.631,-176.114,7.997,148.424
C02578=1198.738,354.340,-75.664,-176.112,8.000,148.424
C02579=1198.734,354.588,-75.696,-176.110,8.003,148.425
C02580=1198.730,354.836,-75.730,-176.108,8.007,148.425
C02581=1198.726,355.084,-75.763,-176.106,8.009,148.425
C02582=1198.721,355.331,-75.796,-176.105,8.013,148.426
C02583=1198.717,355.579,-75.829,-176.102,8.016,148.426
C02584=1198.714,355.827,-75.862,-176.100,8.020,148.426
C02585=1198.710,356.074,-75.895,-176.099,8.022,148.426
C02586=1198.706,356.322,-75.928,-176.097,8.026,148.427
C02587=1198.701,356.570,-75.961,-176.095,8.029,148.427
C02588=1198.697,356.817,-75.994,-176.093,8.032,148.427
C02589=1198.693,357.065,-76.027,-176.091,8.035,148.427
C02590=1198.688,357.313,-76.061,-176.089,8.039,148.428
C02591=1198.684,357.561,-76.094,-176.088,8.041,148.428
C02592=1198.680,357.808,-76.128,-176.086,8.045,148.428
C02593=1198.676,358.056,-76.161,-176.084,8.048,148.429
C02594=1198.672,358.303,-76.194,-176.082,8.051,148.429
C02595=1198.668,358.551,-76.228,-176.080,8.054,148.429
C02596=1198.664,358.800,-76.261,-176.078,8.058,148.430
C02597=1198.660,359.047,-76.294,-176.077,8.061,148.430
C02598=1198.656,359.295,-76.327,-176.074,8.064,148.430
C02599=1198.652,359.543,-76.361,-176.073,8.068,148.431
C02600=1198.648,359.790,-76.394,-176.071,8.070,148.431
C02601=1198.644,360.038,-76.428,-176.069,8.074,148.431
C02602=1198.640,360.285,-76.461,-176.067,8.077,148.431
C02603=1198.636,360.533,-76.494,-176.066,8.080,148.432
C02604=1198.631,360.781,-76.528,-176.064,8.084,148.432
C02605=1198.628,361.029,-76.562,-176.062,8.087,148.433
C02606=1198.623,361.277,-76.595,-176.061,8.090,148.433
C02607=1198.619,361.524,-76.628,-176.058,8.093,148.433
C02608=1198.615,361.772,-76.661,-176.057,8.097,148.434
C02609=1198.611,362.019,-76.695,-176.055,8.099,148.434
C02610=1198.607,362.267,-76.728,-176.053,8.103,148.434
C02611=1198.602,362.515,-76.762,-176.052,8.106,148.435
C02612=1198.599,362.763,-76.796,-176.050,8.109,148.435
C02613=1198.595,363.011,-76.830,-176.048,8.113,148.435
C02614=1198.591,363.258,-76.863,-176.047,8.115,148.436
C02615=1198.587,363.506,-76.896,-176.045,8.119,148.436
C02616=1198.583,363.753,-76.930,-176.043,8.122,148.436
C02617=1198.579,364.002,-76.964,-176.041,8.125,148.437
C02618=1198.575,364.249,-76.998,-176.040,8.128,148.437
C02619=1198.571,364.497,-77.031,-176.038,8.132,148.438
C02620=1198.566,364.744,-77.064,-176.036,8.135,148.438
C02621=1198.562,364.992,-77.098,-176.035,8.138,148.438
C02622=1198.558,365.240,-77.132,-176.033,8.141,148.439
C02623=1198.555,365.487,-77.166,-176.032,8.144,148.439
C02624=1198.550,365.735,-77.199,-176.030,8.148,148.439
C02625=1198.546,365.983,-77.233,-176.028,8.150,148.440
C02626=1198.542,366.263,-77.271,-176.027,8.154,148.440
C02627=1198.537,366.544,-77.309,-176.025,8.158,148.440
C02628=1198.533,366.825,-77.348,-176.023,8.161,148.441
C02629=1198.528,367.107,-77.386,-176.021,8.165,148.441
C02630=1198.524,367.354,-77.420,-176.020,8.168,148.442
C02631=1198.520,367.601,-77.454,-176.018,8.171,148.442
C02632=1198.515,367.849,-77.487,-176.017,8.175,148.443
C02633=1198.512,368.097,-77.522,-176.015,8.178,148.443
C02634=1198.508,368.344,-77.555,-176.014,8.181,148.443
C02635=1198.503,368.592,-77.589,-176.012,8.184,148.444
C02636=1198.499,368.840,-77.622,-176.011,8.188,148.444
C02637=1198.496,369.087,-77.657,-176.009,8.191,148.445
C02638=1198.491,369.335,-77.690,-176.008,8.193,148.445
C02639=1198.487,369.583,-77.724,-176.006,8.197,148.445
C02640=1198.483,369.830,-77.758,-176.005,8.200,148.446
C02641=1198.479,370.078,-77.792,-176.003,8.204,148.446
C02642=1198.475,370.326,-77.826,-176.002,8.206,148.447
C02643=1198.470,370.574,-77.860,-176.001,8.209,148.447
C02644=1198.466,370.821,-77.894,-175.999,8.213,148.448
C02645=1198.463,371.068,-77.928,-175.998,8.216,148.448
C02646=1198.458,371.317,-77.962,-175.996,8.219,148.448
C02647=1198.454,371.564,-77.995,-175.995,8.222,148.449
C02648=1198.450,371.812,-78.030,-175.994,8.225,148.449
C02649=1198.447,372.059,-78.064,-175.992,8.228,148.450
C02650=1198.442,372.307,-78.098,-175.991,8.232,148.450
C02651=1198.439,372.555,-78.132,-175.990,8.234,148.451
C02652=1198.435,372.802,-78.166,-175.988,8.238,148.451
C02653=1198.430,373.050,-78.200,-175.987,8.241,148.451
C02654=1198.427,373.298,-78.234,-175.986,8.244,148.452
C02655=1198.422,373.545,-78.269,-175.984,8.247,148.452
C02656=1198.418,373.792,-78.302,-175.983,8.250,148.453
C02657=1198.414,374.041,-78.336,-175.982,8.253,148.453
C02658=1198.410,374.288,-78.370,-175.980,8.257,148.454
C02659=1198.406,374.535,-78.405,-175.979,8.260,148.454
C02660=1198.402,374.783,-78.439,-175.978,8.263,148.455
C02661=1198.398,375.031,-78.474,-175.977,8.265,148.455
C02662=1198.394,375.278,-78.507,-175.975,8.269,148.455
C02663=1198.390,375.527,-78.542,-175.974,8.272,148.456
C02664=1198.386,375.774,-78.575,-175.973,8.275,148.456
C02665=1198.381,376.021,-78.610,-175.972,8.278,148.457
C02666=1198.378,376.269,-78.644,-175.971,8.282,148.457
C02667=1198.373,376.516,-78.679,-175.969,8.285,148.458
C02668=1198.370,376.763,-78.712,-175.968,8.287,148.458
C02669=1198.366,377.012,-78.747,-175.967,8.290,148.459
C02670=1198.361,377.259,-78.780,-175.966,8.293,148.459
C02671=1198.358,377.507,-78.815,-175.964,8.297,148.460
C02672=1198.353,377.755,-78.850,-175.964,8.300,148.460
C02673=1198.349,378.002,-78.884,-175.962,8.303,148.461
C02674=1198.345,378.250,-78.918,-175.962,8.306,148.461
C02675=1198.341,378.497,-78.952,-175.960,8.309,148.462
C02676=1198.337,378.745,-78.987,-175.960,8.312,148.462
C02677=1198.334,378.992,-79.021,-175.958,8.315,148.463
C02678=1198.329,379.240,-79.055,-175.958,8.318,148.463
C02679=1198.325,379.488,-79.090,-175.956,8.321,148.464
C02680=1198.321,379.735,-79.124,-175.955,8.324,148.464
C02681=1198.317,379.983,-79.159,-175.954,8.327,148.465
C02682=1198.313,380.231,-79.193,-175.953,8.330,148.465
C02683=1198.309,380.478,-79.227,-175.952,8.333,148.466
C02684=1198.305,380.726,-79.262,-175.951,8.336,148.466
C02685=1198.301,380.973,-79.296,-175.950,8.339,148.466
C02686=1198.297,381.221,-79.331,-175.949,8.342,148.467
C02687=1198.292,381.468,-79.365,-175.948,8.345,148.467
C02688=1198.289,381.716,-79.400,-175.947,8.348,148.468
C02689=1198.285,381.964,-79.434,-175.946,8.351,148.469
C02690=1198.280,382.211,-79.469,-175.945,8.354,148.469
C02691=1198.277,382.459,-79.503,-175.944,8.357,148.470
C02692=1198.272,382.706,-79.537,-175.943,8.360,148.470
C02693=1198.269,382.954,-79.573,-175.942,8.363,148.471
C02694=1198.265,383.201,-79.607,-175.941,8.366,148.471
C02695=1198.261,383.449,-79.641,-175.940,8.369,148.472
C02696=1198.256,383.696,-79.676,-175.939,8.372,148.472
C02697=1198.252,383.945,-79.711,-175.939,8.375,148.473
C02698=1198.248,384.192,-79.745,-175.938,8.377,148.473
C02699=1198.244,384.440,-79.779,-175.937,8.380,148.474
C02700=1198.240,384.687,-79.814,-175.936,8.383,148.474
C02701=1198.236,384.934,-79.849,-175.935,8.386,148.475
C02702=1198.232,385.182,-79.883,-175.934,8.389,148.475
C02703=1198.228,385.429,-79.918,-175.934,8.392,148.476
C02704=1198.224,385.677,-79.953,-175.933,8.395,148.476
C02705=1198.220,385.924,-79.987,-175.932,8.397,148.477
C02706=1198.216,386.172,-80.022,-175.931,8.400,148.477
C02707=1198.212,386.419,-80.057,-175.931,8.404,148.478
C02708=1198.208,386.668,-80.091,-175.930,8.407,148.479
C02709=1198.204,386.915,-80.125,-175.929,8.410,148.479
C02710=1198.200,387.163,-80.160,-175.928,8.412,148.479
C02711=1198.196,387.410,-80.195,-175.928,8.415,148.480
C02712=1198.192,387.658,-80.230,-175.927,8.418,148.481
C02713=1198.188,387.905,-80.264,-175.926,8.421,148.481
C02714=1198.184,388.153,-80.299,-175.926,8.423,148.482
C02715=1198.180,388.400,-80.334,-175.925,8.426,148.482
C02716=1198.176,388.648,-80.369,-175.924,8.429,148.483
C02717=1198.172,388.896,-80.404,-175.924,8.432,148.483
C02718=1198.168,389.142,-80.438,-175.923,8.435,148.484
C02719=1198.164,389.391,-80.473,-175.922,8.438,148.484
C02720=1198.160,389.638,-80.508,-175.922,8.440,148.485
C02721=1198.156,389.886,-80.542,-175.921,8.443,148.486
C02722=1198.151,390.133,-80.578,-175.920,8.446,148.486
C02723=1198.148,390.381,-80.612,-175.920,8.448,148.486
C02724=1198.144,390.628,-80.646,-175.919,8.451,148.487
C02725=1198.140,390.876,-80.682,-175.919,8.454,148.488
C02726=1198.135,391.123,-80.716,-175.918,8.457,148.488
C02727=1198.132,391.371,-80.752,-175.917,8.460,148.489
C02728=1198.127,391.618,-80.786,-175.917,8.462,148.489
C02729=1198.124,391.866,-80.821,-175.916,8.465,148.490
C02730=1198.119,392.148,-80.861,-175.915,8.468,148.490
C02731=1198.115,392.432,-80.900,-175.914,8.471,148.491
C02732=1198.110,392.715,-80.941,-175.914,8.474,148.492
C02733=1198.105,392.998,-80.980,-175.913,8.477,148.492
C02734=1198.102,393.245,-81.015,-175.913,8.480,148.493
C02735=1198.097,393.493,-81.050,-175.912,8.482,148.493
C02736=1198.093,393.740,-81.085,-175.912,8.485,148.494
C02737=1198.089,393.988,-81.120,-175.911,8.487,148.494
C02738=1198.085,394.236,-81.155,-175.911,8.491,148.495
C02739=1198.082,394.483,-81.190,-175.910,8.493,148.496
C02740=1198.077,394.730,-81.224,-175.910,8.496,148.496
C02741=1198.074,394.978,-81.260,-175.909,8.498,148.497
C02742=1198.069,395.225,-81.294,-175.909,8.500,148.497
C02743=1198.066,395.473,-81.330,-175.908,8.504,148.498
C02744=1198.062,395.721,-81.365,-175.908,8.506,148.498
C02745=1198.057,395.968,-81.400,-175.907,8.509,148.499
C02746=1198.053,396.216,-81.435,-175.907,8.511,148.499
C02747=1198.049,396.463,-81.470,-175.907,8.513,148.500
C02748=1198.045,396.711,-81.505,-175.906,8.517,148.501
C02749=1198.041,396.958,-81.540,-175.906,8.519,148.501
C02750=1198.037,397.206,-81.575,-175.906,8.521,148.502
C02751=1198.034,397.453,-81.610,-175.905,8.524,148.502
C02752=1198.029,397.700,-81.644,-175.905,8.526,148.503
C02753=1198.026,397.948,-81.680,-175.904,8.529,148.503
C02754=1198.021,398.195,-81.714,-175.904,8.532,148.504
C02755=1198.017,398.443,-81.750,-175.903,8.534,148.504
C02756=1198.014,398.691,-81.784,-175.903,8.536,148.505
C02757=1198.009,398.938,-81.820,-175.903,8.539,148.505
C02758=1198.005,399.186,-81.854,-175.902,8.542,148.506
C02759=1198.002,399.433,-81.890,-175.902,8.544,148.507
C02760=1197.997,399.680,-81.925,-175.902,8.546,148.507
C02761=1197.993,399.928,-81.960,-175.901,8.549,148.508
C02762=1197.989,400.175,-81.995,-175.901,8.552,148.508
C02763=1197.985,400.423,-82.030,-175.900,8.554,148.509
C02764=1197.981,400.671,-82.066,-175.900,8.556,148.509
C02765=1197.977,400.918,-82.100,-175.899,8.558,148.510
C02766=1197.973,401.165,-82.136,-175.899,8.560,148.510
C02767=1197.970,401.413,-82.171,-175.898,8.563,148.511
C02768=1197.965,401.660,-82.206,-175.898,8.566,148.511
C02769=1197.961,401.908,-82.241,-175.898,8.568,148.512
C02770=1197.957,402.155,-82.276,-175.898,8.570,148.512
C02771=1197.953,402.403,-82.311,-175.897,8.573,148.513
C02772=1197.949,402.650,-82.347,-175.897,8.575,148.513
C02773=1197.945,402.898,-82.381,-175.896,8.578,148.514
C02774=1197.941,403.145,-82.417,-175.896,8.580,148.515
C02775=1197.938,403.393,-82.452,-175.896,8.582,148.515
C02776=1197.933,403.640,-82.487,-175.896,8.585,148.516
C02777=1197.929,403.888,-82.522,-175.896,8.587,148.516
C02778=1197.926,404.135,-82.558,-175.895,8.589,148.517
C02779=1197.921,404.383,-82.592,-175.895,8.592,148.517
C02780=1197.917,404.630,-82.628,-175.895,8.594,148.518
C02781=1197.914,404.878,-82.663,-175.895,8.596,148.518
C02782=1197.909,405.125,-82.698,-175.894,8.599,148.519
C02783=1197.906,405.372,-82.733,-175.894,8.601,148.519
C02784=1197.902,405.620,-82.769,-175.893,8.604,148.520
C02785=1197.897,405.867,-82.803,-175.893,8.606,148.520
C02786=1197.894,406.115,-82.839,-175.893,8.608,148.521
C02787=1197.889,406.363,-82.875,-175.893,8.610,148.521
C02788=1197.885,406.610,-82.910,-175.892,8.613,148.522
C02789=1197.881,406.858,-82.945,-175.892,8.615,148.523
C02790=1197.877,407.105,-82.981,-175.892,8.617,148.523
C02791=1197.873,407.352,-83.016,-175.892,8.620,148.524
C02792=1197.869,407.600,-83.051,-175.891,8.622,148.524
C02793=1197.865,407.848,-83.086,-175.891,8.624,148.525
C02794=1197.861,408.094,-83.121,-175.891,8.626,148.525
C02795=1197.858,408.342,-83.157,-175.891,8.629,148.526
C02796=1197.854,408.590,-83.192,-175.891,8.631,148.526
C02797=1197.850,408.837,-83.227,-175.890,8.633,148.527
C02798=1197.846,409.084,-83.263,-175.890,8.635,148.527
C02799=1197.842,409.332,-83.298,-175.889,8.637,148.528
C02800=1197.838,409.580,-83.334,-175.889,8.640,148.528
C02801=1197.833,409.827,-83.369,-175.889,8.642,148.529
C02802=1197.829,410.075,-83.404,-175.889,8.643,148.529
C02803=1197.826,410.322,-83.440,-175.889,8.646,148.530
C02804=1197.821,410.569,-83.475,-175.889,8.648,148.530
C02805=1197.817,410.817,-83.510,-175.889,8.650,148.531
C02806=1197.814,411.064,-83.545,-175.888,8.652,148.531
C02807=1197.810,411.312,-83.581,-175.888,8.655,148.532
C02808=1197.806,411.559,-83.616,-175.888,8.657,148.532
C02809=1197.801,411.807,-83.652,-175.888,8.659,148.533
C02810=1197.798,412.054,-83.688,-175.887,8.661,148.533
C02811=1197.793,412.301,-83.722,-175.887,8.663,148.534
C02812=1197.790,412.549,-83.758,-175.887,8.665,148.534
C02813=1197.786,412.796,-83.793,-175.887,8.667,148.535
C02814=1197.782,413.044,-83.829,-175.887,8.669,148.535
C02815=1197.778,413.291,-83.864,-175.886,8.672,148.536
C02816=1197.774,413.539,-83.900,-175.886,8.674,148.536
C02817=1197.770,413.787,-83.935,-175.886,8.676,148.537
C02818=1197.765,414.033,-83.970,-175.885,8.678,148.537
C02819=1197.762,414.281,-84.006,-175.885,8.680,148.538
C02820=1197.758,414.528,-84.041,-175.885,8.682,148.538
C02821=1197.754,414.776,-84.077,-175.885,8.684,148.539
C02822=1197.750,415.023,-84.112,-175.885,8.686,148.539
C02823=1197.746,415.271,-84.148,-175.884,8.689,148.540
C02824=1197.742,415.519,-84.183,-175.884,8.691,148.540
C02825=1197.738,415.766,-84.219,-175.884,8.692,148.540
C02826=1197.733,416.101,-84.267,-175.884,8.695,148.541
C02827=1197.728,416.436,-84.315,-175.884,8.698,148.542
C02828=1197.728,416.771,-84.362,-175.883,8.701,148.543
C02829=1197.730,417.105,-84.409,-175.883,8.703,148.543
C02830=1197.309,417.106,-84.449,-175.886,8.714,148.547
C02831=1197.307,416.769,-84.401,-175.886,8.712,148.546
C02832=1197.307,416.430,-84.353,-175.887,8.708,148.545
C02833=1197.311,416.093,-84.304,-175.887,8.706,148.545
C02834=1197.317,415.755,-84.256,-175.887,8.703,148.544
C02835=1197.320,415.507,-84.220,-175.887,8.702,148.544
C02836=1197.325,415.260,-84.186,-175.888,8.699,148.543
C02837=1197.329,415.012,-84.150,-175.888,8.697,148.543
C02838=1197.332,414.765,-84.115,-175.888,8.695,148.542
C02839=1197.336,414.517,-84.079,-175.888,8.693,148.542
C02840=1197.341,414.270,-84.043,-175.888,8.691,148.541
C02841=1197.344,414.023,-84.008,-175.888,8.689,148.541
C02842=1197.348,413.775,-83.972,-175.889,8.687,148.540
C02843=1197.352,413.528,-83.937,-175.889,8.685,148.540
C02844=1197.356,413.280,-83.902,-175.889,8.682,148.539
C02845=1197.360,413.033,-83.867,-175.890,8.680,148.539
C02846=1197.364,412.785,-83.830,-175.890,8.678,148.538
C02847=1197.369,412.538,-83.795,-175.890,8.676,148.538
C02848=1197.372,412.291,-83.760,-175.890,8.674,148.537
C02849=1197.376,412.043,-83.724,-175.890,8.672,148.537
C02850=1197.380,411.796,-83.689,-175.890,8.670,148.536
C02851=1197.384,411.548,-83.654,-175.891,8.667,148.536
C02852=1197.388,411.301,-83.619,-175.891,8.665,148.535
C02853=1197.392,411.053,-83.582,-175.891,8.663,148.535
C02854=1197.397,410.806,-83.547,-175.892,8.661,148.534
C02855=1197.400,410.559,-83.512,-175.892,8.659,148.534
C02856=1197.404,410.311,-83.477,-175.892,8.657,148.533
C02857=1197.408,410.063,-83.441,-175.892,8.655,148.533
C02858=1197.412,409.816,-83.406,-175.892,8.653,148.532
C02859=1197.416,409.569,-83.371,-175.892,8.650,148.532
C02860=1197.419,409.321,-83.335,-175.893,8.648,148.531
C02861=1197.424,409.074,-83.301,-175.893,8.646,148.531
C02862=1197.428,408.826,-83.265,-175.893,8.644,148.530
C02863=1197.432,408.579,-83.229,-175.893,8.641,148.530
C02864=1197.436,408.331,-83.193,-175.894,8.639,148.529
C02865=1197.440,408.084,-83.159,-175.894,8.637,148.529
C02866=1197.444,407.836,-83.123,-175.894,8.634,148.528
C02867=1197.448,407.589,-83.088,-175.894,8.632,148.528
C02868=1197.452,407.342,-83.053,-175.894,8.630,148.527
C02869=1197.456,407.094,-83.018,-175.895,8.628,148.527
C02870=1197.460,406.846,-82.982,-175.895,8.626,148.526
C02871=1197.464,406.599,-82.947,-175.896,8.623,148.526
C02872=1197.468,406.352,-82.911,-175.896,8.621,148.525
C02873=1197.471,406.104,-82.877,-175.896,8.619,148.525
C02874=1197.476,405.857,-82.841,-175.896,8.617,148.524
C02875=1197.479,405.610,-82.806,-175.897,8.614,148.524
C02876=1197.484,405.361,-82.770,-175.897,8.612,148.523
C02877=1197.488,405.114,-82.735,-175.897,8.610,148.522
C02878=1197.492,404.867,-82.700,-175.897,8.608,148.522
C02879=1197.496,404.619,-82.664,-175.897,8.605,148.521
C02880=1197.500,404.372,-82.630,-175.898,8.603,148.521
C02881=1197.504,404.124,-82.594,-175.899,8.600,148.520
C02882=1197.508,403.877,-82.559,-175.899,8.598,148.520
C02883=1197.512,403.629,-82.524,-175.899,8.595,148.519
C02884=1197.516,403.382,-82.489,-175.899,8.593,148.519
C02885=1197.519,403.134,-82.453,-175.899,8.591,148.518
C02886=1197.524,402.887,-82.419,-175.900,8.589,148.518
C02887=1197.528,402.640,-82.383,-175.900,8.586,148.517
C02888=1197.531,402.392,-82.348,-175.900,8.584,148.517
C02889=1197.536,402.145,-82.313,-175.900,8.582,148.516
C02890=1197.540,401.897,-82.278,-175.901,8.579,148.516
C02891=1197.544,401.649,-82.243,-175.901,8.576,148.515
C02892=1197.548,401.402,-82.208,-175.902,8.574,148.514
C02893=1197.552,401.155,-82.172,-175.902,8.572,148.514
C02894=1197.555,400.907,-82.137,-175.902,8.570,148.513
C02895=1197.560,400.660,-82.102,-175.903,8.567,148.513
C02896=1197.564,400.412,-82.067,-175.903,8.564,148.512
C02897=1197.568,400.165,-82.032,-175.903,8.562,148.512
C02898=1197.572,399.917,-81.996,-175.904,8.560,148.511
C02899=1197.576,399.669,-81.962,-175.904,8.557,148.511
C02900=1197.580,399.422,-81.926,-175.905,8.554,148.510
C02901=1197.584,399.174,-81.892,-175.905,8.552,148.510
C02902=1197.587,398.927,-81.856,-175.905,8.550,148.509
C02903=1197.592,398.680,-81.821,-175.905,8.548,148.508
C02904=1197.596,398.432,-81.786,-175.906,8.544,148.508
C02905=1197.600,398.185,-81.751,-175.906,8.542,148.507
C02906=1197.604,397.937,-81.716,-175.907,8.540,148.507
C02907=1197.608,397.690,-81.680,-175.907,8.537,148.506
C02908=1197.612,397.442,-81.646,-175.908,8.535,148.506
C02909=1197.616,397.195,-81.610,-175.908,8.532,148.505
C02910=1197.620,396.947,-81.576,-175.909,8.529,148.505
C02911=1197.623,396.700,-81.541,-175.909,8.527,148.504
C02912=1197.627,396.452,-81.506,-175.909,8.525,148.504
C02913=1197.632,396.205,-81.471,-175.910,8.522,148.503
C02914=1197.636,395.957,-81.436,-175.910,8.519,148.502
C02915=1197.640,395.710,-81.401,-175.910,8.517,148.502
C02916=1197.644,395.462,-81.366,-175.911,8.514,148.501
C02917=1197.647,395.215,-81.331,-175.911,8.512,148.501
C02918=1197.652,394.967,-81.296,-175.912,8.509,148.500
C02919=1197.656,394.720,-81.261,-175.912,8.506,148.500
C02920=1197.660,394.472,-81.226,-175.913,8.504,148.499
C02921=1197.664,394.225,-81.191,-175.913,8.501,148.499
C02922=1197.668,393.977,-81.156,-175.914,8.499,148.498
C02923=1197.672,393.729,-81.122,-175.914,8.496,148.497
C02924=1197.675,393.482,-81.086,-175.915,8.493,148.497
C02925=1197.680,393.235,-81.052,-175.915,8.490,148.496
C02926=1197.684,392.987,-81.016,-175.916,8.488,148.496
C02927=1197.688,392.704,-80.977,-175.916,8.485,148.495
C02928=1197.693,392.421,-80.937,-175.917,8.482,148.495
C02929=1197.697,392.138,-80.897,-175.918,8.479,148.494
C02930=1197.702,391.855,-80.857,-175.919,8.475,148.493
C02931=1197.706,391.607,-80.822,-175.919,8.473,148.493
C02932=1197.710,391.360,-80.787,-175.920,8.470,148.492
C02933=1197.714,391.112,-80.753,-175.921,8.467,148.492
C02934=1197.718,390.865,-80.718,-175.921,8.465,148.491
C02935=1197.722,390.617,-80.683,-175.922,8.462,148.491
C02936=1197.726,390.370,-80.648,-175.922,8.459,148.490
C02937=1197.730,390.122,-80.613,-175.923,8.456,148.489
C02938=1197.735,389.875,-80.578,-175.923,8.453,148.489
C02939=1197.738,389.627,-80.544,-175.924,8.451,148.488
C02940=1197.742,389.379,-80.509,-175.925,8.448,148.488
C02941=1197.746,389.132,-80.474,-175.925,8.446,148.487
C02942=1197.750,388.884,-80.439,-175.926,8.443,148.487
C02943=1197.755,388.637,-80.405,-175.927,8.440,148.486
C02944=1197.758,388.390,-80.370,-175.927,8.436,148.486
C02945=1197.762,388.142,-80.335,-175.928,8.434,148.485
C02946=1197.766,387.894,-80.300,-175.928,8.431,148.485
C02947=1197.771,387.647,-80.266,-175.930,8.428,148.484
C02948=1197.774,387.399,-80.230,-175.930,8.426,148.484
C02949=1197.778,387.152,-80.196,-175.931,8.423,148.483
C02950=1197.782,386.904,-80.162,-175.931,8.420,148.482
C02951=1197.787,386.656,-80.127,-175.932,8.417,148.482
C02952=1197.790,386.409,-80.092,-175.933,8.414,148.481
C02953=1197.794,386.162,-80.058,-175.934,8.412,148.481
C02954=1197.798,385.914,-80.023,-175.934,8.409,148.480
C02955=1197.803,385.666,-79.988,-175.935,8.405,148.480
C02956=1197.807,385.418,-79.954,-175.936,8.403,148.479
C02957=1197.810,385.172,-79.919,-175.937,8.400,148.479
C02958=1197.814,384.924,-79.884,-175.937,8.397,148.478
C02959=1197.819,384.676,-79.850,-175.938,8.394,148.478
C02960=1197.823,384.428,-79.815,-175.939,8.391,148.477
C02961=1197.827,384.181,-79.781,-175.940,8.388,148.477
C02962=1197.831,383.933,-79.746,-175.941,8.385,148.476
C02963=1197.835,383.686,-79.711,-175.942,8.382,148.475
C02964=1197.838,383.438,-79.677,-175.943,8.379,148.475
C02965=1197.843,383.191,-79.642,-175.944,8.376,148.474
C02966=1197.847,382.943,-79.608,-175.945,8.373,148.474
C02967=1197.850,382.696,-79.574,-175.946,8.370,148.474
C02968=1197.855,382.448,-79.539,-175.947,8.367,148.473
C02969=1197.859,382.200,-79.504,-175.948,8.364,148.473
C02970=1197.863,381.953,-79.470,-175.949,8.361,148.472
C02971=1197.867,381.705,-79.436,-175.949,8.358,148.471
C02972=1197.871,381.458,-79.400,-175.951,8.355,148.471
C02973=1197.874,381.210,-79.366,-175.951,8.352,148.470
C02974=1197.879,380.963,-79.332,-175.953,8.349,148.470
C02975=1197.883,380.715,-79.297,-175.953,8.346,148.469
C02976=1197.887,380.468,-79.263,-175.954,8.343,148.469
C02977=1197.891,380.220,-79.229,-175.955,8.340,148.468
C02978=1197.895,379.972,-79.194,-175.956,8.337,148.468
C02979=1197.899,379.725,-79.160,-175.957,8.335,148.467
C02980=1197.903,379.477,-79.125,-175.958,8.331,148.467
C02981=1197.908,379.229,-79.091,-175.959,8.329,148.466
C02982=1197.911,378.982,-79.057,-175.960,8.326,148.466
C02983=1197.915,378.734,-79.022,-175.961,8.323,148.466
C02984=1197.919,378.487,-78.988,-175.963,8.319,148.465
C02985=1197.923,378.239,-78.953,-175.964,8.316,148.464
C02986=1197.928,377.991,-78.919,-175.965,8.313,148.464
C02987=1197.932,377.744,-78.885,-175.966,8.310,148.463
C02988=1197.936,377.496,-78.851,-175.967,8.307,148.463
C02989=1197.940,377.249,-78.817,-175.968,8.304,148.463
C02990=1197.944,377.001,-78.782,-175.970,8.301,148.462
C02991=1197.948,376.753,-78.748,-175.971,8.298,148.462
C02992=1197.952,376.506,-78.714,-175.972,8.295,148.461
C02993=1197.955,376.258,-78.679,-175.973,8.292,148.461
C02994=1197.960,376.011,-78.645,-175.974,8.289,148.460
C02995=1197.964,375.763,-78.610,-175.976,8.285,148.460
C02996=1197.968,375.515,-78.576,-175.977,8.282,148.459
C02997=1197.973,375.267,-78.542,-175.978,8.279,148.459
C02998=1197.976,375.020,-78.509,-175.979,8.276,148.458
C02999=1197.980,374.772,-78.474,-175.981,8.273,148.458
C03000=1197.984,374.525,-78.440,-175.982,8.270,148.457
C03001=1197.988,374.277,-78.405,-175.983,8.267,148.457
C03002=1197.992,374.030,-78.371,-175.984,8.264,148.457
C03003=1197.997,373.782,-78.337,-175.986,8.260,148.456
C03004=1198.000,373.534,-78.303,-175.987,8.258,148.456
C03005=1198.004,373.287,-78.269,-175.988,8.254,148.455
C03006=1198.009,373.039,-78.235,-175.989,8.251,148.455
C03007=1198.012,372.791,-78.201,-175.991,8.248,148.454
C03008=1198.017,372.544,-78.167,-175.992,8.245,148.454
C03009=1198.020,372.296,-78.133,-175.994,8.242,148.453
C03010=1198.025,372.049,-78.099,-175.995,8.239,148.453
C03011=1198.029,371.801,-78.065,-175.996,8.236,148.452
C03012=1198.033,371.553,-78.031,-175.997,8.232,148.452
C03013=1198.037,371.306,-77.997,-175.999,8.229,148.452
C03014=1198.040,371.058,-77.963,-176.000,8.226,148.451
C03015=1198.045,370.810,-77.929,-176.002,8.223,148.451
C03016=1198.049,370.563,-77.895,-176.003,8.220,148.450
C03017=1198.053,370.314,-77.861,-176.005,8.216,148.450
C03018=1198.057,370.067,-77.827,-176.006,8.214,148.450
C03019=1198.061,369.820,-77.793,-176.008,8.210,148.449
C03020=1198.066,369.572,-77.759,-176.009,8.207,148.449
C03021=1198.069,369.324,-77.725,-176.011,8.204,148.448
C03022=1198.074,369.076,-77.691,-176.012,8.201,148.448
C03023=1198.078,368.829,-77.657,-176.013,8.198,148.448
C03024=1198.081,368.582,-77.623,-176.015,8.194,148.447
C03025=1198.086,368.333,-77.589,-176.016,8.191,148.447
C03026=1198.090,368.086,-77.555,-176.018,8.188,148.446
C03027=1198.094,367.838,-77.522,-176.019,8.185,148.446
C03028=1198.098,367.591,-77.488,-176.021,8.181,148.445
C03029=1198.102,367.343,-77.454,-176.022,8.179,148.445
C03030=1198.106,367.096,-77.420,-176.024,8.175,148.445
C03031=1198.110,366.815,-77.382,-176.026,8.171,148.444
C03032=1198.115,366.534,-77.344,-176.027,8.168,148.444
C03033=1198.120,366.253,-77.306,-176.029,8.164,148.443
C03034=1198.125,365.972,-77.267,-176.031,8.160,148.443
C03035=1198.128,365.724,-77.234,-176.033,8.158,148.443
C03036=1198.132,365.477,-77.200,-176.034,8.154,148.442
C03037=1198.136,365.229,-77.167,-176.036,8.151,148.442
C03038=1198.141,364.982,-77.132,-176.037,8.148,148.441
C03039=1198.145,364.733,-77.099,-176.039,8.145,148.441
C03040=1198.149,364.486,-77.066,-176.041,8.142,148.441
C03041=1198.153,364.238,-77.032,-176.043,8.138,148.440
C03042=1198.157,363.991,-76.998,-176.044,8.135,148.440
C03043=1198.161,363.743,-76.964,-176.046,8.132,148.440
C03044=1198.165,363.495,-76.931,-176.047,8.129,148.439
C03045=1198.169,363.247,-76.897,-176.049,8.125,148.439
C03046=1198.173,363.000,-76.863,-176.051,8.122,148.439
C03047=1198.177,362.752,-76.830,-176.053,8.119,148.438
C03048=1198.182,362.504,-76.797,-176.054,8.116,148.438
C03049=1198.186,362.257,-76.763,-176.056,8.113,148.438
C03050=1198.189,362.009,-76.729,-176.058,8.110,148.437
C03051=1198.193,361.761,-76.696,-176.060,8.106,148.437
C03052=1198.197,361.513,-76.663,-176.061,8.103,148.436
C03053=1198.201,361.266,-76.629,-176.063,8.100,148.436
C03054=1198.206,361.018,-76.595,-176.065,8.096,148.436
C03055=1198.210,360.770,-76.562,-176.066,8.094,148.436
C03056=1198.214,360.523,-76.529,-176.068,8.090,148.435
C03057=1198.218,360.275,-76.495,-176.069,8.087,148.435
C03058=1198.222,360.027,-76.462,-176.072,8.084,148.435
C03059=1198.226,359.779,-76.428,-176.073,8.080,148.434
C03060=1198.230,359.532,-76.395,-176.075,8.078,148.434
C03061=1198.234,359.284,-76.362,-176.077,8.074,148.434
C03062=1198.238,359.037,-76.328,-176.079,8.071,148.433
C03063=1198.242,358.789,-76.295,-176.080,8.068,148.433
C03064=1198.247,358.541,-76.261,-176.083,8.065,148.433
C03065=1198.251,358.293,-76.228,-176.084,8.061,148.432
C03066=1198.255,358.046,-76.195,-176.087,8.058,148.432
C03067=1198.259,357.797,-76.161,-176.088,8.055,148.432
C03068=1198.263,357.549,-76.128,-176.090,8.051,148.431
C03069=1198.267,357.302,-76.095,-176.092,8.048,148.431
C03070=1198.271,357.054,-76.062,-176.093,8.045,148.431
C03071=1198.275,356.806,-76.029,-176.096,8.042,148.431
C03072=1198.279,356.559,-75.996,-176.097,8.038,148.430
C03073=1198.284,356.311,-75.963,-176.099,8.036,148.430
C03074=1198.288,356.063,-75.929,-176.101,8.033,148.430
C03075=1198.292,355.816,-75.895,-176.103,8.029,148.429
C03076=1198.296,355.568,-75.863,-176.105,8.026,148.429
C03077=1198.300,355.320,-75.830,-176.107,8.023,148.429
C03078=1198.304,355.072,-75.797,-176.109,8.019,148.428
C03079=1198.308,354.824,-75.764,-176.111,8.016,148.428
C03080=1198.313,354.577,-75.730,-176.113,8.014,148.428
C03081=1198.317,354.329,-75.697,-176.114,8.010,148.428
C03082=1198.321,354.081,-75.664,-176.117,8.007,148.427
C03083=1198.324,353.834,-75.632,-176.118,8.004,148.427
C03084=1198.328,353.586,-75.598,-176.121,8.001,148.427
C03085=1198.333,353.338,-75.565,-176.122,7.997,148.427
C03086=1198.337,353.091,-75.532,-176.125,7.994,148.426
C03087=1198.341,352.843,-75.499,-176.126,7.991,148.426
C03088=1198.345,352.595,-75.466,-176.129,7.988,148.426
C03089=1198.349,352.347,-75.433,-176.130,7.984,148.425
C03090=1198.354,352.099,-75.400,-176.132,7.982,148.425
C03091=1198.358,351.851,-75.367,-176.134,7.978,148.425
C03092=1198.362,351.604,-75.334,-176.136,7.975,148.425
C03093=1198.365,351.356,-75.301,-176.139,7.972,148.425
C03094=1198.370,351.108,-75.269,-176.140,7.969,148.424
C03095=1198.374,350.860,-75.236,-176.142,7.966,148.424
C03096=1198.378,350.612,-75.203,-176.144,7.962,148.424
C03097=1198.382,350.365,-75.169,-176.146,7.960,148.424
C03098=1198.387,350.116,-75.137,-176.148,7.957,148.423
C03099=1198.390,349.869,-75.104,-176.150,7.953,148.423
C03100=1198.394,349.621,-75.071,-176.152,7.950,148.423
C03101=1198.399,349.373,-75.039,-176.154,7.947,148.423
C03102=1198.403,349.125,-75.006,-176.156,7.944,148.422
C03103=1198.407,348.877,-74.972,-176.158,7.940,148.422
C03104=1198.411,348.630,-74.941,-176.161,7.937,148.422
C03105=1198.415,348.382,-74.908,-176.162,7.935,148.422
C03106=1198.419,348.135,-74.875,-176.165,7.931,148.421
C03107=1198.424,347.886,-74.842,-176.167,7.928,148.421
C03108=1198.427,347.639,-74.810,-176.168,7.925,148.421
C03109=1198.431,347.391,-74.777,-176.171,7.922,148.421
C03110=1198.436,347.143,-74.744,-176.173,7.919,148.421
C03111=1198.440,346.895,-74.711,-176.175,7.915,148.420
C03112=1198.444,346.647,-74.679,-176.177,7.913,148.420
C03113=1198.448,346.399,-74.646,-176.179,7.910,148.420
C03114=1198.453,346.152,-74.614,-176.181,7.906,148.420
C03115=1198.457,345.904,-74.581,-176.182,7.903,148.419
C03116=1198.461,345.656,-74.549,-176.185,7.900,148.419
C03117=1198.465,345.408,-74.516,-176.187,7.897,148.419
C03118=1198.469,345.160,-74.483,-176.190,7.894,148.419
C03119=1198.473,344.912,-74.451,-176.191,7.891,148.419
C03120=1198.478,344.665,-74.419,-176.193,7.888,148.419
C03121=1198.482,344.417,-74.385,-176.196,7.885,148.418
C03122=1198.486,344.169,-74.354,-176.198,7.881,148.418
C03123=1198.490,343.921,-74.320,-176.200,7.879,148.418
C03124=1198.494,343.673,-74.288,-176.202,7.875,148.418
C03125=1198.498,343.425,-74.255,-176.204,7.872,148.417
C03126=1198.503,343.178,-74.223,-176.206,7.869,148.417
C03127=1198.506,342.930,-74.192,-176.208,7.866,148.417
C03128=1198.510,342.682,-74.158,-176.210,7.863,148.417
C03129=1198.515,342.434,-74.126,-176.212,7.860,148.417
C03130=1198.519,342.186,-74.094,-176.214,7.857,148.416
C03131=1198.523,341.939,-74.061,-176.216,7.854,148.416
C03132=1198.527,341.691,-74.029,-176.219,7.851,148.416
C03133=1198.531,341.442,-73.997,-176.221,7.847,148.416
C03134=1198.535,341.195,-73.964,-176.223,7.845,148.416
C03135=1198.540,340.916,-73.929,-176.226,7.841,148.416
C03136=1198.545,340.638,-73.892,-176.228,7.837,148.415
C03137=1198.549,340.359,-73.856,-176.230,7.834,148.415
C03138=1198.554,340.081,-73.820,-176.233,7.831,148.415
C03139=1198.559,339.833,-73.787,-176.235,7.828,148.415
C03140=1198.562,339.585,-73.755,-176.237,7.824,148.415
C03141=1198.567,339.337,-73.723,-176.239,7.822,148.415
C03142=1198.571,339.090,-73.691,-176.241,7.818,148.414
C03143=1198.575,338.842,-73.658,-176.243,7.815,148.414
C03144=1198.579,338.594,-73.626,-176.246,7.812,148.414
C03145=1198.583,338.345,-73.594,-176.248,7.810,148.414
C03146=1198.588,338.098,-73.563,-176.250,7.806,148.414
C03147=1198.591,337.850,-73.531,-176.252,7.803,148.413
C03148=1198.596,337.602,-73.498,-176.255,7.800,148.413
C03149=1198.599,337.354,-73.466,-176.257,7.797,148.413
C03150=1198.604,337.106,-73.434,-176.259,7.794,148.413
C03151=1198.608,336.858,-73.402,-176.261,7.791,148.413
C03152=1198.612,336.610,-73.369,-176.263,7.789,148.413
C03153=1198.617,336.363,-73.338,-176.265,7.785,148.413
C03154=1198.620,336.115,-73.306,-176.268,7.782,148.412
C03155=1198.625,335.866,-73.274,-176.270,7.779,148.412
C03156=1198.629,335.619,-73.242,-176.272,7.776,148.412
C03157=1198.633,335.371,-73.210,-176.274,7.773,148.412
C03158=1198.637,335.123,-73.178,-176.276,7.770,148.412
C03159=1198.642,334.875,-73.146,-176.279,7.767,148.412
C03160=1198.646,334.627,-73.114,-176.281,7.764,148.412
C03161=1198.650,334.379,-73.082,-176.283,7.761,148.411
C03162=1198.654,334.131,-73.051,-176.286,7.758,148.411
C03163=1198.658,333.883,-73.019,-176.288,7.754,148.411
C03164=1198.662,333.635,-72.986,-176.290,7.752,148.411
C03165=1198.667,333.388,-72.955,-176.292,7.749,148.411
C03166=1198.670,333.140,-72.923,-176.295,7.746,148.411
C03167=1198.675,332.891,-72.891,-176.297,7.742,148.411
C03168=1198.679,332.643,-72.860,-176.299,7.740,148.411
C03169=1198.683,332.395,-72.828,-176.301,7.737,148.410
C03170=1198.688,332.148,-72.796,-176.304,7.734,148.410
C03171=1198.692,331.900,-72.764,-176.305,7.731,148.410
C03172=1198.695,331.652,-72.732,-176.308,7.728,148.410
C03173=1198.700,331.404,-72.701,-176.310,7.725,148.410
C03174=1198.705,331.155,-72.669,-176.313,7.721,148.410
C03175=1198.709,330.908,-72.637,-176.315,7.719,148.410
C03176=1198.713,330.660,-72.606,-176.317,7.716,148.410
C03177=1198.716,330.412,-72.574,-176.319,7.713,148.409
C03178=1198.721,330.165,-72.542,-176.322,7.710,148.409
C03179=1198.725,329.916,-72.511,-176.324,7.707,148.409
C03180=1198.730,329.668,-72.479,-176.326,7.704,148.409
C03181=1198.733,329.420,-72.447,-176.328,7.701,148.409
C03182=1198.738,329.172,-72.416,-176.331,7.698,148.409
C03183=1198.742,328.924,-72.385,-176.333,7.695,148.409
C03184=1198.745,328.676,-72.353,-176.336,7.692,148.409
C03185=1198.751,328.428,-72.321,-176.338,7.689,148.409
C03186=1198.754,328.180,-72.290,-176.339,7.686,148.409
C03187=1198.759,327.933,-72.258,-176.342,7.683,148.409
C03188=1198.763,327.684,-72.227,-176.344,7.680,148.408
C03189=1198.767,327.437,-72.195,-176.347,7.677,148.408
C03190=1198.771,327.189,-72.164,-176.349,7.674,148.408
C03191=1198.775,326.941,-72.133,-176.351,7.671,148.408
C03192=1198.779,326.693,-72.101,-176.354,7.668,148.408
C03193=1198.784,326.445,-72.070,-176.356,7.665,148.408
C03194=1198.788,326.196,-72.038,-176.358,7.663,148.408
C03195=1198.793,325.948,-72.007,-176.361,7.660,148.408
C03196=1198.796,325.700,-71.975,-176.363,7.656,148.408
C03197=1198.801,325.453,-71.944,-176.365,7.654,148.408
C03198=1198.805,325.204,-71.913,-176.368,7.651,148.408
C03199=1198.809,324.957,-71.881,-176.370,7.648,148.407
C03200=1198.813,324.708,-71.850,-176.373,7.645,148.407
C03201=1198.818,324.460,-71.819,-176.374,7.642,148.407
C03202=1198.821,324.212,-71.787,-176.377,7.639,148.407
C03203=1198.826,323.964,-71.757,-176.379,7.636,148.407
C03204=1198.830,323.716,-71.725,-176.382,7.633,148.407
C03205=1198.834,323.468,-71.694,-176.384,7.630,148.407
C03206=1198.839,323.221,-71.663,-176.386,7.627,148.407
C03207=1198.843,322.972,-71.631,-176.389,7.624,148.407
C03208=1198.847,322.724,-71.601,-176.391,7.622,148.407
C03209=1198.851,322.476,-71.569,-176.393,7.619,148.407
C03210=1198.856,322.228,-71.538,-176.396,7.615,148.406
C03211=1198.859,321.981,-71.507,-176.398,7.612,148.406
C03212=1198.863,321.733,-71.476,-176.400,7.610,148.407
C03213=1198.868,321.485,-71.445,-176.403,7.607,148.406
C03214=1198.872,321.237,-71.413,-176.405,7.604,148.406
C03215=1198.876,320.989,-71.383,-176.408,7.601,148.406
C03216=1198.880,320.740,-71.352,-176.410,7.598,148.406
C03217=1198.885,320.492,-71.321,-176.412,7.595,148.406
C03218=1198.889,320.245,-71.289,-176.415,7.592,148.406
C03219=1198.893,319.996,-71.258,-176.417,7.590,148.406
C03220=1198.898,319.748,-71.227,-176.419,7.587,148.406
C03221=1198.901,319.500,-71.197,-176.422,7.583,148.406
C03222=1198.905,319.252,-71.165,-176.424,7.580,148.406
C03223=1198.910,319.004,-71.135,-176.426,7.578,148.406
C03224=1198.914,318.756,-71.103,-176.429,7.575,148.406
C03225=1198.918,318.508,-71.073,-176.431,7.572,148.406
C03226=1198.923,318.260,-71.042,-176.433,7.570,148.406
C03227=1198.926,318.012,-71.011,-176.436,7.566,148.405
C03228=1198.931,317.764,-70.980,-176.438,7.563,148.405
C03229=1198.935,317.516,-70.949,-176.441,7.560,148.405
C03230=1198.939,317.268,-70.918,-176.443,7.558,148.406
C03231=1198.944,317.020,-70.887,-176.445,7.555,148.405
C03232=1198.948,316.772,-70.857,-176.448,7.552,148.405
C03233=1198.952,316.523,-70.826,-176.450,7.549,148.405
C03234=1198.956,316.275,-70.795,-176.453,7.546,148.405
C03235=1198.961,316.027,-70.764,-176.455,7.543,148.405
C03236=1198.964,315.779,-70.734,-176.458,7.540,148.405
C03237=1198.969,315.531,-70.703,-176.460,7.538,148.405
C03238=1198.974,315.283,-70.672,-176.462,7.535,148.405
C03239=1198.978,315.007,-70.638,-176.465,7.532,148.405
C03240=1198.983,314.730,-70.604,-176.468,7.529,148.405
C03241=1198.988,314.454,-70.570,-176.470,7.525,148.405
C03242=1198.992,314.178,-70.535,-176.473,7.522,148.405
C03243=1198.996,313.930,-70.504,-176.475,7.519,148.405
C03244=1199.000,313.682,-70.474,-176.478,7.516,148.405
C03245=1199.005,313.434,-70.444,-176.481,7.513,148.405
C03246=1199.009,313.185,-70.413,-176.483,7.511,148.405
C03247=1199.013,312.937,-70.383,-176.485,7.508,148.405
C03248=1199.018,312.689,-70.352,-176.488,7.505,148.405
C03249=1199.022,312.442,-70.321,-176.490,7.502,148.405
C03250=1199.026,312.193,-70.291,-176.493,7.499,148.405
C03251=1199.030,311.945,-70.260,-176.495,7.496,148.405
C03252=1199.034,311.698,-70.230,-176.497,7.494,148.405
C03253=1199.039,311.449,-70.200,-176.500,7.491,148.405
C03254=1199.043,311.200,-70.169,-176.502,7.488,148.405
C03255=1199.047,310.953,-70.139,-176.505,7.485,148.405
C03256=1199.051,310.705,-70.108,-176.507,7.483,148.405
C03257=1199.056,310.456,-70.078,-176.509,7.479,148.405
C03258=1199.060,310.209,-70.048,-176.512,7.476,148.405
C03259=1199.065,309.961,-70.017,-176.514,7.474,148.405
C03260=1199.068,309.712,-69.986,-176.517,7.471,148.405
C03261=1199.073,309.464,-69.956,-176.520,7.468,148.405
C03262=1199.077,309.216,-69.926,-176.522,7.466,148.405
C03263=1199.082,308.968,-69.895,-176.524,7.462,148.404
C03264=1199.086,308.720,-69.866,-176.527,7.459,148.404
C03265=1199.090,308.472,-69.835,-176.529,7.457,148.405
C03266=1199.094,308.223,-69.805,-176.531,7.454,148.405
C03267=1199.099,307.975,-69.775,-176.534,7.451,148.405
C03268=1199.102,307.727,-69.744,-176.536,7.449,148.405
C03269=1199.107,307.479,-69.714,-176.538,7.446,148.404
C03270=1199.111,307.231,-69.684,-176.541,7.443,148.404
C03271=1199.116,306.983,-69.653,-176.543,7.440,148.405
C03272=1199.120,306.735,-69.624,-176.546,7.437,148.405
C03273=1199.124,306.486,-69.593,-176.549,7.434,148.405
C03274=1199.128,306.238,-69.563,-176.551,7.432,148.405
C03275=1199.132,305.990,-69.533,-176.554,7.429,148.405
C03276=1199.137,305.742,-69.502,-176.556,7.426,148.405
C03277=1199.141,305.494,-69.473,-176.558,7.424,148.405
C03278=1199.145,305.246,-69.442,-176.561,7.421,148.404
C03279=1199.150,304.998,-69.413,-176.563,7.418,148.404
C03280=1199.154,304.750,-69.383,-176.566,7.415,148.405
C03281=1199.158,304.502,-69.353,-176.568,7.412,148.405
C03282=1199.163,304.253,-69.323,-176.571,7.409,148.405
C03283=1199.167,304.005,-69.292,-176.574,7.406,148.405
C03284=1199.171,303.757,-69.263,-176.576,7.404,148.405
C03285=1199.175,303.509,-69.232,-176.578,7.401,148.405
C03286=1199.180,303.260,-69.202,-176.580,7.399,148.405
C03287=1199.184,303.012,-69.172,-176.583,7.396,148.405
C03288=1199.188,302.764,-69.143,-176.586,7.393,148.405
C03289=1199.193,302.516,-69.113,-176.588,7.390,148.405
C03290=1199.196,302.268,-69.082,-176.590,7.387,148.405
C03291=1199.201,302.020,-69.053,-176.593,7.384,148.405
C03292=1199.206,301.771,-69.023,-176.595,7.382,148.405
C03293=1199.209,301.523,-68.993,-176.598,7.379,148.405
C03294=1199.214,301.275,-68.963,-176.600,7.376,148.405
C03295=1199.218,301.027,-68.934,-176.603,7.374,148.405
C03296=1199.222,300.779,-68.903,-176.605,7.371,148.405
C03297=1199.227,300.531,-68.874,-176.608,7.368,148.405
C03298=1199.231,300.282,-68.844,-176.610,7.366,148.405
C03299=1199.235,300.034,-68.815,-176.613,7.363,148.405
C03300=1199.240,299.786,-68.785,-176.616,7.360,148.405
C03301=1199.244,299.538,-68.755,-176.618,7.358,148.405
C03302=1199.248,299.290,-68.725,-176.620,7.355,148.405
C03303=1199.252,299.041,-68.696,-176.623,7.352,148.405
C03304=1199.256,298.793,-68.666,-176.625,7.349,148.405
C03305=1199.261,298.545,-68.636,-176.628,7.346,148.405
C03306=1199.265,298.297,-68.606,-176.630,7.344,148.405
C03307=1199.269,298.049,-68.577,-176.633,7.341,148.405
C03308=1199.273,297.800,-68.547,-176.635,7.338,148.405
C03309=1199.278,297.552,-68.518,-176.638,7.336,148.405
C03310=1199.282,297.305,-68.489,-176.640,7.333,148.405
C03311=1199.287,297.056,-68.458,-176.643,7.330,148.405
C03312=1199.292,296.808,-68.429,-176.645,7.328,148.405
C03313=1199.296,296.559,-68.400,-176.648,7.325,148.405
C03314=1199.300,296.311,-68.370,-176.650,7.322,148.405
C03315=1199.304,296.063,-68.341,-176.653,7.320,148.405
C03316=1199.308,295.815,-68.311,-176.655,7.317,148.406
C03317=1199.312,295.566,-68.282,-176.657,7.314,148.406
C03318=1199.316,295.319,-68.252,-176.660,7.311,148.406
C03319=1199.321,295.070,-68.223,-176.663,7.308,148.406
C03320=1199.325,294.822,-68.193,-176.665,7.306,148.406
C03321=1199.329,294.573,-68.164,-176.668,7.303,148.406
C03322=1199.334,294.326,-68.135,-176.670,7.300,148.406
C03323=1199.338,294.077,-68.105,-176.673,7.298,148.406
C03324=1199.343,293.829,-68.075,-176.675,7.295,148.406
C03325=1199.347,293.581,-68.046,-176.677,7.293,148.406
C03326=1199.351,293.332,-68.016,-176.681,7.290,148.406
C03327=1199.356,293.084,-67.987,-176.683,7.287,148.406
C03328=1199.360,292.836,-67.958,-176.685,7.285,148.406
C03329=1199.364,292.588,-67.928,-176.688,7.282,148.406
C03330=1199.369,292.340,-67.899,-176.690,7.280,148.406
C03331=1199.373,292.091,-67.871,-176.693,7.277,148.406
C03332=1199.377,291.843,-67.841,-176.696,7.274,148.406
C03333=1199.381,291.595,-67.812,-176.698,7.271,148.406
C03334=1199.385,291.347,-67.782,-176.700,7.268,148.406
C03335=1199.389,291.098,-67.753,-176.703,7.266,148.407
C03336=1199.394,290.850,-67.725,-176.705,7.263,148.407
C03337=1199.399,290.602,-67.695,-176.708,7.260,148.407
C03338=1199.403,290.354,-67.666,-176.710,7.258,148.407
C03339=1199.407,290.105,-67.636,-176.713,7.255,148.407
C03340=1199.411,289.856,-67.608,-176.715,7.253,148.407
C03341=1199.416,289.609,-67.578,-176.718,7.250,148.407
C03342=1199.420,289.361,-67.549,-176.721,7.247,148.407
C03343=1199.425,289.086,-67.517,-176.724,7.244,148.407
C03344=1199.429,288.812,-67.485,-176.726,7.241,148.407
C03345=1199.435,288.537,-67.452,-176.729,7.238,148.407
C03346=1199.439,288.263,-67.421,-176.732,7.236,148.407
C03347=1199.444,288.015,-67.391,-176.734,7.233,148.407
C03348=1199.447,287.767,-67.362,-176.737,7.230,148.407
C03349=1199.452,287.518,-67.334,-176.739,7.228,148.407
C03350=1199.456,287.270,-67.305,-176.742,7.225,148.407
C03351=1199.461,287.021,-67.276,-176.744,7.223,148.408
C03352=1199.466,286.774,-67.247,-176.747,7.220,148.408
C03353=1199.470,286.525,-67.218,-176.750,7.217,148.408
C03354=1199.473,286.277,-67.189,-176.752,7.215,148.408
C03355=1199.478,286.029,-67.160,-176.755,7.212,148.408
C03356=1199.483,285.780,-67.131,-176.757,7.210,148.408
C03357=1199.487,285.532,-67.102,-176.759,7.207,148.408
C03358=1199.491,285.284,-67.074,-176.762,7.204,148.408
C03359=1199.495,285.036,-67.045,-176.765,7.202,148.408
C03360=1199.500,284.787,-67.016,-176.767,7.199,148.408
C03361=1199.504,284.539,-66.987,-176.770,7.197,148.408
C03362=1199.508,284.290,-66.958,-176.772,7.194,148.408
C03363=1199.513,284.042,-66.930,-176.774,7.191,148.409
C03364=1199.517,283.794,-66.901,-176.777,7.188,148.409
C03365=1199.522,283.545,-66.872,-176.780,7.186,148.409
C03366=1199.526,283.298,-66.843,-176.782,7.183,148.409
C03367=1199.530,283.049,-66.815,-176.785,7.181,148.409
C03368=1199.535,282.800,-66.786,-176.787,7.178,148.409
C03369=1199.539,282.553,-66.757,-176.790,7.175,148.409
C03370=1199.543,282.304,-66.729,-176.792,7.173,148.409
C03371=1199.548,282.056,-66.700,-176.795,7.170,148.409
C03372=1199.552,281.808,-66.671,-176.798,7.168,148.409
C03373=1199.556,281.559,-66.643,-176.800,7.165,148.409
C03374=1199.561,281.310,-66.614,-176.802,7.163,148.410
C03375=1199.565,281.063,-66.585,-176.805,7.160,148.410
C03376=1199.569,280.814,-66.557,-176.808,7.158,148.410
C03377=1199.574,280.566,-66.529,-176.810,7.155,148.410
C03378=1199.578,280.318,-66.499,-176.813,7.153,148.410
C03379=1199.582,280.070,-66.472,-176.815,7.150,148.410
C03380=1199.587,279.821,-66.443,-176.817,7.148,148.410
C03381=1199.591,279.572,-66.414,-176.821,7.145,148.410
C03382=1199.595,279.324,-66.386,-176.823,7.142,148.410
C03383=1199.600,279.076,-66.357,-176.825,7.140,148.410
C03384=1199.604,278.828,-66.329,-176.828,7.137,148.410
C03385=1199.608,278.579,-66.300,-176.831,7.135,148.411
C03386=1199.612,278.330,-66.272,-176.833,7.132,148.411
C03387=1199.617,278.082,-66.244,-176.836,7.130,148.411
C03388=1199.621,277.834,-66.215,-176.838,7.127,148.411
C03389=1199.626,277.586,-66.187,-176.840,7.125,148.411
C03390=1199.630,277.337,-66.159,-176.844,7.122,148.411
C03391=1199.635,277.089,-66.130,-176.846,7.120,148.411
C03392=1199.638,276.841,-66.102,-176.848,7.117,148.411
C03393=1199.643,276.592,-66.073,-176.851,7.115,148.411
C03394=1199.647,276.344,-66.046,-176.854,7.112,148.412
C03395=1199.652,276.095,-66.017,-176.856,7.110,148.412
C03396=1199.656,275.847,-65.989,-176.859,7.107,148.412
C03397=1199.661,275.598,-65.960,-176.861,7.105,148.412
C03398=1199.665,275.350,-65.933,-176.864,7.102,148.412
C03399=1199.669,275.102,-65.904,-176.866,7.100,148.412
C03400=1199.674,274.854,-65.876,-176.869,7.097,148.412
C03401=1199.678,274.605,-65.848,-176.871,7.095,148.413
C03402=1199.683,274.357,-65.819,-176.874,7.092,148.413
C03403=1199.686,274.108,-65.791,-176.876,7.090,148.413
C03404=1199.691,273.860,-65.763,-176.879,7.087,148.413
C03405=1199.695,273.612,-65.735,-176.882,7.085,148.413
C03406=1199.700,273.364,-65.707,-176.884,7.082,148.413
C03407=1199.704,273.115,-65.678,-176.886,7.080,148.413
C03408=1199.708,272.867,-65.651,-176.889,7.077,148.413
C03409=1199.713,272.619,-65.623,-176.892,7.075,148.413
C03410=1199.718,272.370,-65.595,-176.894,7.072,148.413
C03411=1199.722,272.122,-65.567,-176.897,7.069,148.414
C03412=1199.726,271.873,-65.539,-176.900,7.067,148.414
C03413=1199.731,271.625,-65.510,-176.902,7.065,148.414
C03414=1199.734,271.376,-65.482,-176.905,7.062,148.414
C03415=1199.739,271.128,-65.455,-176.907,7.059,148.414
C03416=1199.744,270.879,-65.427,-176.910,7.057,148.414
C03417=1199.748,270.631,-65.399,-176.912,7.055,148.414
C03418=1199.752,270.383,-65.371,-176.915,7.052,148.414
C03419=1199.756,270.135,-65.343,-176.917,7.050,148.415
C03420=1199.761,269.886,-65.315,-176.920,7.048,148.415
C03421=1199.765,269.637,-65.287,-176.922,7.045,148.415
C03422=1199.770,269.389,-65.259,-176.925,7.043,148.415
C03423=1199.774,269.141,-65.231,-176.928,7.040,148.415
C03424=1199.779,268.892,-65.203,-176.930,7.037,148.415
C03425=1199.783,268.644,-65.176,-176.933,7.035,148.415
C03426=1199.787,268.396,-65.148,-176.935,7.033,148.416
C03427=1199.791,268.147,-65.120,-176.938,7.030,148.416
C03428=1199.797,267.899,-65.092,-176.940,7.028,148.416
C03429=1199.800,267.650,-65.064,-176.943,7.025,148.416
C03430=1199.805,267.402,-65.037,-176.945,7.023,148.416
C03431=1199.809,267.154,-65.009,-176.948,7.021,148.416
C03432=1199.813,266.905,-64.982,-176.951,7.018,148.416
C03433=1199.818,266.657,-64.954,-176.953,7.016,148.416
C03434=1199.823,266.409,-64.926,-176.956,7.013,148.417
C03435=1199.827,266.159,-64.898,-176.958,7.011,148.417
C03436=1199.831,265.912,-64.870,-176.961,7.008,148.417
C03437=1199.836,265.663,-64.843,-176.963,7.006,148.417
C03438=1199.840,265.414,-64.815,-176.966,7.003,148.417
C03439=1199.844,265.166,-64.788,-176.968,7.001,148.417
C03440=1199.849,264.918,-64.760,-176.971,6.999,148.418
C03441=1199.853,264.669,-64.732,-176.974,6.996,148.418
C03442=1199.858,264.421,-64.704,-176.976,6.994,148.418
C03443=1199.862,264.172,-64.677,-176.979,6.991,148.418
C03444=1199.866,263.924,-64.649,-176.981,6.989,148.418
C03445=1199.871,263.675,-64.622,-176.984,6.986,148.418
C03446=1199.875,263.427,-64.594,-176.986,6.984,148.418
C03447=1199.881,263.154,-64.565,-176.990,6.981,148.419
C03448=1199.885,262.881,-64.535,-176.992,6.979,148.419
C03449=1199.890,262.608,-64.504,-176.995,6.976,148.419
C03450=1199.894,262.336,-64.475,-176.998,6.973,148.419
C03451=1199.898,262.088,-64.447,-177.000,6.971,148.419
C03452=1199.903,261.839,-64.420,-177.003,6.968,148.419
C03453=1199.908,261.591,-64.392,-177.005,6.966,148.419
C03454=1199.912,261.343,-64.365,-177.008,6.964,148.420
C03455=1199.916,261.093,-64.337,-177.010,6.961,148.420
C03456=1199.921,260.845,-64.310,-177.013,6.959,148.420
C03457=1199.925,260.597,-64.282,-177.016,6.957,148.420
C03458=1199.930,260.349,-64.255,-177.018,6.954,148.420
C03459=1199.934,260.099,-64.228,-177.021,6.952,148.420
C03460=1199.938,259.851,-64.201,-177.023,6.950,148.421
C03461=1199.943,259.603,-64.173,-177.025,6.947,148.421
C03462=1199.947,259.355,-64.146,-177.029,6.945,148.421
C03463=1199.952,259.106,-64.119,-177.031,6.942,148.421
C03464=1199.956,258.857,-64.092,-177.034,6.940,148.421
C03465=1199.961,258.608,-64.064,-177.036,6.938,148.421
C03466=1199.965,258.360,-64.037,-177.039,6.936,148.422
C03467=1199.970,258.112,-64.010,-177.041,6.933,148.422
C03468=1199.974,257.863,-63.983,-177.043,6.931,148.422
C03469=1199.978,257.615,-63.956,-177.047,6.928,148.422
C03470=1199.982,257.366,-63.929,-177.049,6.926,148.422
C03471=1199.987,257.118,-63.902,-177.051,6.924,148.422
C03472=1199.991,256.870,-63.874,-177.054,6.921,148.423
C03473=1199.996,256.621,-63.847,-177.057,6.919,148.423
C03474=1200.001,256.373,-63.820,-177.059,6.917,148.423
C03475=1200.005,256.125,-63.793,-177.062,6.914,148.423
C03476=1200.009,255.875,-63.766,-177.064,6.912,148.423
C03477=1200.013,255.627,-63.739,-177.067,6.909,148.423
C03478=1200.018,255.378,-63.712,-177.070,6.907,148.424
C03479=1200.023,255.130,-63.685,-177.072,6.905,148.424
C03480=1200.027,254.881,-63.658,-177.075,6.902,148.424
C03481=1200.031,254.633,-63.631,-177.077,6.900,148.424
C03482=1200.036,254.385,-63.604,-177.080,6.898,148.424
C03483=1200.040,254.136,-63.577,-177.082,6.895,148.424
C03484=1200.045,253.888,-63.550,-177.085,6.893,148.425
C03485=1200.048,253.639,-63.523,-177.087,6.891,148.425
C03486=1200.053,253.390,-63.496,-177.090,6.888,148.425
C03487=1200.058,253.142,-63.469,-177.093,6.886,148.425
C03488=1200.062,252.893,-63.442,-177.095,6.884,148.425
C03489=1200.066,252.645,-63.415,-177.098,6.882,148.426
C03490=1200.071,252.397,-63.388,-177.100,6.879,148.426
C03491=1200.076,252.148,-63.361,-177.103,6.878,148.426
C03492=1200.080,251.899,-63.336,-177.105,6.875,148.426
C03493=1200.085,251.651,-63.309,-177.108,6.873,148.426
C03494=1200.089,251.402,-63.281,-177.110,6.871,148.426
C03495=1200.093,251.154,-63.255,-177.113,6.868,148.427
C03496=1200.098,250.906,-63.228,-177.116,6.866,148.427
C03497=1200.102,250.657,-63.201,-177.118,6.864,148.427
C03498=1200.107,250.408,-63.175,-177.121,6.861,148.427
C03499=1200.111,250.160,-63.148,-177.123,6.859,148.427
C03500=1200.116,249.911,-63.121,-177.126,6.857,148.428
C03501=1200.120,249.663,-63.095,-177.129,6.854,148.428
C03502=1200.125,249.415,-63.067,-177.131,6.852,148.428
C03503=1200.129,249.166,-63.041,-177.134,6.850,148.428
C03504=1200.133,248.917,-63.015,-177.136,6.847,148.428
C03505=1200.138,248.669,-62.988,-177.139,6.845,148.429
C03506=1200.142,248.420,-62.962,-177.141,6.843,148.429
C03507=1200.147,248.172,-62.935,-177.144,6.840,148.429
C03508=1200.151,247.923,-62.908,-177.146,6.838,148.429
C03509=1200.156,247.675,-62.881,-177.149,6.836,148.429
C03510=1200.160,247.426,-62.855,-177.152,6.833,148.429
C03511=1200.164,247.178,-62.828,-177.154,6.832,148.430
C03512=1200.169,246.928,-62.802,-177.157,6.829,148.430
C03513=1200.173,246.680,-62.776,-177.160,6.827,148.430
C03514=1200.178,246.432,-62.749,-177.162,6.825,148.430
C03515=1200.182,246.183,-62.723,-177.165,6.823,148.431
C03516=1200.187,245.935,-62.696,-177.167,6.821,148.431
C03517=1200.191,245.686,-62.669,-177.170,6.818,148.431
C03518=1200.196,245.437,-62.643,-177.173,6.816,148.431
C03519=1200.200,245.189,-62.616,-177.175,6.814,148.431
C03520=1200.205,244.940,-62.590,-177.178,6.811,148.432
C03521=1200.209,244.692,-62.564,-177.180,6.809,148.432
C03522=1200.213,244.443,-62.537,-177.183,6.807,148.432
C03523=1200.217,244.194,-62.511,-177.185,6.804,148.432
C03524=1200.222,243.945,-62.485,-177.188,6.802,148.432
C03525=1200.227,243.698,-62.458,-177.190,6.800,148.432
C03526=1200.231,243.449,-62.433,-177.193,6.798,148.433
C03527=1200.236,243.201,-62.406,-177.196,6.796,148.433
C03528=1200.240,242.952,-62.380,-177.198,6.793,148.433
C03529=1200.245,242.703,-62.353,-177.201,6.792,148.433
C03530=1200.249,242.454,-62.327,-177.203,6.789,148.434
C03531=1200.253,242.206,-62.301,-177.206,6.787,148.434
C03532=1200.258,241.957,-62.274,-177.208,6.785,148.434
C03533=1200.262,241.708,-62.248,-177.211,6.783,148.434
C03534=1200.267,241.461,-62.222,-177.214,6.780,148.435
C03535=1200.271,241.212,-62.196,-177.216,6.778,148.435
C03536=1200.276,240.963,-62.170,-177.219,6.776,148.435
C03537=1200.280,240.714,-62.143,-177.221,6.774,148.435
C03538=1200.285,240.466,-62.117,-177.224,6.771,148.435
C03539=1200.289,240.217,-62.092,-177.227,6.769,148.436
C03540=1200.293,239.968,-62.065,-177.229,6.767,148.436
C03541=1200.298,239.720,-62.039,-177.232,6.765,148.436
C03542=1200.302,239.471,-62.014,-177.234,6.762,148.436
C03543=1200.307,239.223,-61.986,-177.237,6.761,148.436
C03544=1200.311,238.974,-61.961,-177.239,6.758,148.437
C03545=1200.316,238.725,-61.935,-177.242,6.757,148.437
C03546=1200.320,238.477,-61.910,-177.245,6.754,148.437
C03547=1200.325,238.229,-61.882,-177.247,6.752,148.437
C03548=1200.329,237.980,-61.857,-177.250,6.750,148.438
C03549=1200.334,237.731,-61.831,-177.252,6.748,148.438
C03550=1200.338,237.482,-61.805,-177.255,6.745,148.438
C03551=1200.343,237.211,-61.776,-177.258,6.743,148.438
C03552=1200.348,236.939,-61.748,-177.261,6.741,148.439
C03553=1200.353,236.668,-61.719,-177.263,6.738,148.439
C03554=1200.358,236.397,-61.692,-177.266,6.736,148.439
C03555=1200.362,236.148,-61.666,-177.269,6.734,148.439
C03556=1200.367,235.899,-61.640,-177.271,6.732,148.439
C03557=1200.371,235.650,-61.614,-177.274,6.730,148.440
C03558=1200.376,235.402,-61.589,-177.277,6.727,148.440
C03559=1200.380,235.153,-61.563,-177.279,6.725,148.440
C03560=1200.384,234.905,-61.536,-177.282,6.723,148.440
C03561=1200.388,234.656,-61.511,-177.284,6.721,148.441
C03562=1200.394,234.408,-61.485,-177.287,6.718,148.441
C03563=1200.398,234.159,-61.459,-177.290,6.717,148.441
C03564=1200.402,233.910,-61.433,-177.292,6.715,148.441
C03565=1200.407,233.662,-61.408,-177.295,6.713,148.442
C03566=1200.412,233.413,-61.382,-177.298,6.710,148.442
C03567=1200.416,233.165,-61.356,-177.300,6.708,148.442
C03568=1200.420,232.916,-61.330,-177.303,6.706,148.442
C03569=1200.425,232.668,-61.305,-177.305,6.704,148.443
C03570=1200.430,232.419,-61.279,-177.307,6.702,148.443
C03571=1200.434,232.170,-61.253,-177.311,6.699,148.443
C03572=1200.439,231.922,-61.228,-177.313,6.697,148.443
C03573=1200.443,231.673,-61.202,-177.315,6.695,148.443
C03574=1200.448,231.423,-61.177,-177.318,6.693,148.444
C03575=1200.452,231.175,-61.151,-177.321,6.692,148.444
C03576=1200.457,230.927,-61.126,-177.323,6.689,148.444
C03577=1200.461,230.678,-61.100,-177.326,6.687,148.444
C03578=1200.466,230.430,-61.075,-177.329,6.685,148.445
C03579=1200.470,230.181,-61.049,-177.331,6.683,148.445
C03580=1200.474,229.932,-61.023,-177.333,6.681,148.445
C03581=1200.479,229.684,-60.998,-177.337,6.678,148.445
C03582=1200.483,229.435,-60.973,-177.339,6.676,148.446
C03583=1200.488,229.186,-60.947,-177.341,6.674,148.446
C03584=1200.493,228.938,-60.921,-177.344,6.672,148.446
C03585=1200.497,228.689,-60.896,-177.347,6.671,148.447
C03586=1200.502,228.441,-60.870,-177.349,6.668,148.447
C03587=1200.506,228.191,-60.845,-177.352,6.666,148.447
C03588=1200.510,227.942,-60.820,-177.355,6.664,148.447
C03589=1200.515,227.694,-60.794,-177.357,6.662,148.447
C03590=1200.519,227.446,-60.768,-177.359,6.660,148.448
C03591=1200.525,227.197,-60.744,-177.362,6.658,148.448
C03592=1200.529,226.948,-60.718,-177.365,6.655,148.448
C03593=1200.533,226.699,-60.692,-177.367,6.653,148.448
C03594=1200.537,226.451,-60.668,-177.370,6.651,148.449
C03595=1200.542,226.202,-60.642,-177.373,6.650,148.449
C03596=1200.546,225.954,-60.617,-177.375,6.647,148.449
C03597=1200.551,225.705,-60.592,-177.378,6.645,148.449
C03598=1200.556,225.456,-60.567,-177.381,6.643,148.450
C03599=1200.560,225.208,-60.541,-177.383,6.641,148.450
C03600=1200.565,224.958,-60.516,-177.386,6.639,148.450
C03601=1200.569,224.710,-60.490,-177.388,6.637,148.451
C03602=1200.573,224.461,-60.466,-177.391,6.635,148.451
C03603=1200.578,224.213,-60.441,-177.394,6.632,148.451
C03604=1200.582,223.964,-60.415,-177.396,6.630,148.451
C03605=1200.587,223.715,-60.390,-177.399,6.629,148.452
C03606=1200.592,223.467,-60.364,-177.401,6.627,148.452
C03607=1200.597,223.218,-60.340,-177.404,6.625,148.452
C03608=1200.600,222.969,-60.315,-177.406,6.623,148.452
C03609=1200.605,222.721,-60.290,-177.409,6.621,148.453
C03610=1200.610,222.472,-60.264,-177.412,6.618,148.453
C03611=1200.615,222.223,-60.240,-177.414,6.616,148.453
C03612=1200.619,221.974,-60.214,-177.417,6.614,148.453
C03613=1200.623,221.726,-60.190,-177.420,6.612,148.454
C03614=1200.627,221.477,-60.164,-177.422,6.611,148.454
C03615=1200.633,221.228,-60.139,-177.424,6.608,148.454
C03616=1200.637,220.979,-60.114,-177.428,6.606,148.455
C03617=1200.641,220.731,-60.089,-177.430,6.604,148.455
C03618=1200.646,220.482,-60.064,-177.433,6.602,148.455
C03619=1200.651,220.234,-60.039,-177.435,6.600,148.455
C03620=1200.654,219.984,-60.015,-177.438,6.598,148.456
C03621=1200.659,219.736,-59.989,-177.440,6.596,148.456
C03622=1200.664,219.488,-59.965,-177.443,6.594,148.456
C03623=1200.668,219.239,-59.940,-177.446,6.591,148.456
C03624=1200.673,218.990,-59.915,-177.448,6.590,148.457
C03625=1200.677,218.741,-59.890,-177.451,6.588,148.457
C03626=1200.682,218.493,-59.866,-177.454,6.586,148.457
C03627=1200.686,218.244,-59.840,-177.456,6.584,148.458
C03628=1200.691,217.995,-59.815,-177.458,6.582,148.458
C03629=1200.695,217.746,-59.791,-177.461,6.580,148.458
C03630=1200.700,217.498,-59.765,-177.464,6.578,148.458
C03631=1200.705,217.249,-59.741,-177.467,6.576,148.459
C03632=1200.709,217.000,-59.716,-177.470,6.574,148.459
C03633=1200.714,216.751,-59.692,-177.472,6.572,148.459
C03634=1200.717,216.503,-59.666,-177.474,6.570,148.460
C03635=1200.723,216.254,-59.642,-177.477,6.568,148.460
C03636=1200.728,216.005,-59.617,-177.480,6.566,148.460
C03637=1200.731,215.756,-59.593,-177.482,6.564,148.461
C03638=1200.737,215.507,-59.568,-177.485,6.561,148.461
C03639=1200.741,215.260,-59.543,-177.488,6.560,148.461
C03640=1200.745,215.010,-59.518,-177.490,6.558,148.461
C03641=1200.750,214.762,-59.494,-177.493,6.556,148.462
C03642=1200.754,214.512,-59.469,-177.496,6.554,148.462
C03643=1200.759,214.264,-59.444,-177.498,6.552,148.462
C03644=1200.764,214.015,-59.420,-177.500,6.550,148.462
C03645=1200.768,213.766,-59.395,-177.503,6.548,148.463
C03646=1200.773,213.517,-59.371,-177.506,6.546,148.463
C03647=1200.777,213.269,-59.346,-177.509,6.544,148.463
C03648=1200.781,213.020,-59.321,-177.512,6.542,148.464
C03649=1200.786,212.772,-59.297,-177.514,6.540,148.464
C03650=1200.791,212.523,-59.273,-177.516,6.538,148.464
